KUKA KRL program: EPS_2_25694_BP02_A_20251117072356.src

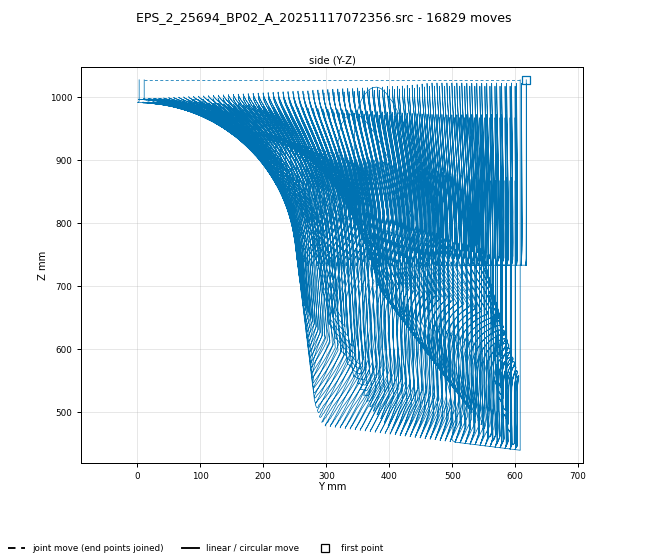
[picture p0: tool path of EPS_2_25694_BP02_A_20251117072356.src, 16829 of 16831 moves have a stored position in this frame; points joined in program order, loops and branches not executed]
&ACCESS RVP
&REL 4
&COMMENT QRS 19112012
&PARAM EDITMASK = *
DEF PART()
EXT BAS (BAS_COMMAND :IN,REAL :IN )
INT I
BAS (#INITMOV,0 )

;KUKA QRS Post kuka4.cps  Date:22-06-2017 !

File_ID=2911

QRS_PRE_INIT()

;Init var - Until changes are made in qrs_pre_init
Outlet_Square_prg=0
Inlet_1_Square_prg=0
Inlet_2_Square_prg=0
Inlet_3_Square_prg=0
Inlet_4_Square_prg=0
Inlet_5_Square_prg=0

Outlet_1={X 0.000, Y 466.000, Z 789.500, B 0.000, E1 0.000 }
Inlet_1={X 0.000, Y 466.000, Z 739.500, B 0.000, E1 180.000 }
Inlet_2={X 0.000, Y 537.940, Z 362.500, B 0.000, E1 273.000 }
Outlet_1_type=457
Inlet_1_type=457
Inlet_2_type=251
;QRS#1=Sidecore dimensions
;QRS#2=450-18" Concrete
;QRS#3=450-18" Concrete
;QRS#4=250-10" PVC SDR 35
;QRS#5=
;QRS#6=
;QRS#7=
;QRS#8=
;QRS#9=28A PSX-2
;QRS#10=28A PSX-2
;QRS#11=14M PSX
;QRS#12=
;QRS#13=
;QRS#14=
;QRS#15=
;QRS#16=1220x127x1372 4,5'
;QRS#17=EPS Height
;QRS#18=1018
;QRS#19=*
;QRS#20= UPDATED VERSION 22-06-2017
;QRS#21=*
Outlet_Square=0250
Inlet_1_Square=0250
Inlet_2_Square=0100
Inlet_3_Square=0
Inlet_4_Square=0
Inlet_5_Square=0
Mill_Square=1
Outlet_Square_Prg=274
Inlet_1_Square_prg=274
Inlet_2_Square_prg=205

QRS_INIT()

$ADVANCE=5

; T1
PTP {E1 171.215,E2 171.215}
PTP {X 0,Y 617.568,A -85,B 0,C 180,E1 171.215,E2 171.215,E3 0,E4 0,E5 0,E6 0}
QRS_SPEED_INIT()
LIN {X 0,Y 617.568,Z 1028,A -85,B 0,C 180,E1 171.215,E2 171.215,E3 0,E4 0,E5 0,E6 0} C_VEL
LIN {X 0,Y 617.568,Z 735.66,A -85,B 0,C 180,E1 171.215,E2 171.215} C_VEL
LIN {X 0,Y 617.546,Z 733.66,A -85,B 0,C 180,E1 171.401,E2 171.401} C_VEL
LIN {X 0,Y 617.995,Z 733.66,A -85,B 0,C 180,E1 174.214,E2 174.214} C_VEL
LIN {X 0,Y 618.056,Z 733.66,A -85,B 0,C 180,E1 178.845,E2 178.845} C_VEL
LIN {X 0,Y 618.024,Z 733.66,A -85,B 0,C 180,E1 183.468,E2 183.468} C_VEL
LIN {X 0,Y 618.034,Z 733.66,A -85,B 0,C 180,E1 188.114,E2 188.114} C_VEL
LIN {X 0,Y 618.015,Z 733.66,A -85,B 0,C 180,E1 192.815,E2 192.815} C_VEL
LIN {X 0,Y 617.991,Z 733.66,A -85,B 0,C 180,E1 197.606,E2 197.606} C_VEL
LIN {X 0,Y 617.8,Z 733.66,A -85,B 0,C 180,E1 198.557,E2 198.557} C_VEL
LIN {X 0,Y 617.948,Z 733.66,A -85,B 0,C 180,E1 202.529,E2 202.529} C_VEL
LIN {X 0,Y 617.447,Z 733.66,A -85,B 0,C 180,E1 205.076,E2 205.076} C_VEL
LIN {X 0,Y 617.888,Z 733.66,A -85,B 0,C 180,E1 207.636,E2 207.636} C_VEL
LIN {X 0,Y 617.379,Z 733.66,A -85,B 0,C 180,E1 210.305,E2 210.305} C_VEL
LIN {X 0,Y 617.845,Z 733.66,A -85,B 0,C 180,E1 212.995,E2 212.995} C_VEL
LIN {X 0,Y 617.716,Z 733.66,A -85,B 0,C 180,E1 214.198,E2 214.198} C_VEL
LIN {X 0,Y 617.779,Z 733.66,A -85,B 0,C 180,E1 218.705,E2 218.705} C_VEL
LIN {X 0,Y 617.447,Z 733.66,A -85,B 0,C 180,E1 221.76,E2 221.76} C_VEL
LIN {X 0,Y 617.88,Z 733.66,A -85,B 0,C 180,E1 224.901,E2 224.901} C_VEL
LIN {X 0,Y 617.778,Z 733.66,A -85,B 0,C 180,E1 228.274,E2 228.274} C_VEL
LIN {X 0,Y 617.563,Z 733.66,A -85,B 0,C 180,E1 231.279,E2 231.279} C_VEL
LIN {X 0,Y 617.589,Z 733.66,A -85,B 0,C 180,E1 231.899,E2 231.899} C_VEL
LIN {X 0,Y 617.834,Z 733.66,A -85,B 0,C 180,E1 234.203,E2 234.203} C_VEL
LIN {X 0,Y 617.355,Z 733.66,A -85,B 0,C 180,E1 236.976,E2 236.976} C_VEL
LIN {X 0,Y 617.906,Z 733.66,A -85,B 0,C 180,E1 239.724,E2 239.724} C_VEL
LIN {X 0,Y 617.897,Z 733.66,A -85,B 0,C 180,E1 243.987,E2 243.987} C_VEL
LIN {X 0,Y 617.787,Z 733.66,A -85,B 0,C 180,E1 244.426,E2 244.426} C_VEL
LIN {X 0,Y 617.131,Z 733.66,A -85,B 0,C 180,E1 244.544,E2 244.544} C_VEL
LIN {X 0,Y 616.404,Z 733.66,A -85,B 0,C 180,E1 244.615,E2 244.615} C_VEL
LIN {X 0,Y 617.534,Z 739.849,A -85,B 0,C 180,E1 244.745,E2 244.745} C_VEL
LIN {X 0,Y 617.679,Z 744.384,A -85,B 0,C 180,E1 244.809,E2 244.809} C_VEL
LIN {X 0,Y 617.925,Z 800.182,A -85,B 0,C 180,E1 245.528,E2 245.528} C_VEL
LIN {X 0,Y 617.874,Z 810.032,A -85,B 0,C 180,E1 245.684,E2 245.684} C_VEL
LIN {X 0,Y 617.799,Z 819.999,A -85,B 0,C 180,E1 245.88,E2 245.88} C_VEL
LIN {X 0,Y 617.89,Z 833.169,A -85,B 0,C 180,E1 246.218,E2 246.218} C_VEL
LIN {X 0,Y 617.827,Z 843.59,A -85,B 0,C 180,E1 246.528,E2 246.528} C_VEL
LIN {X 0,Y 617.931,Z 855.912,A -85,B 0,C 180,E1 246.969,E2 246.969} C_VEL
LIN {X 0,Y 617.951,Z 866.365,A -85,B 0,C 180,E1 247.393,E2 247.393} C_VEL
LIN {X 0,Y 617.873,Z 876.668,A -85,B 0,C 180,E1 247.859,E2 247.859} C_VEL
LIN {X 0,Y 617.944,Z 887.338,A -85,B 0,C 180,E1 248.406,E2 248.406} C_VEL
LIN {X 0,Y 617.966,Z 898.213,A -85,B 0,C 180,E1 249.027,E2 249.027} C_VEL
LIN {X 0,Y 617.938,Z 908.022,A -85,B 0,C 180,E1 249.643,E2 249.643} C_VEL
LIN {X 0,Y 617.949,Z 917.528,A -85,B 0,C 180,E1 250.301,E2 250.301} C_VEL
LIN {X 0,Y 617.957,Z 926.721,A -85,B 0,C 180,E1 250.999,E2 250.999} C_VEL
LIN {X 0,Y 617.963,Z 935.648,A -85,B 0,C 180,E1 251.739,E2 251.739} C_VEL
LIN {X 0,Y 617.942,Z 944.029,A -85,B 0,C 180,E1 252.497,E2 252.497} C_VEL
LIN {X 0,Y 617.896,Z 951.424,A -85,B 0,C 180,E1 253.221,E2 253.221} C_VEL
LIN {X 0,Y 617.949,Z 959.127,A -85,B 0,C 180,E1 254.046,E2 254.046} C_VEL
LIN {X 0,Y 617.972,Z 965.662,A -85,B 0,C 180,E1 254.803,E2 254.803} C_VEL
LIN {X 0,Y 617.889,Z 972.774,A -85,B 0,C 180,E1 255.697,E2 255.697} C_VEL
LIN {X 0,Y 617.879,Z 979.238,A -85,B 0,C 180,E1 256.589,E2 256.589} C_VEL
LIN {X 0,Y 617.985,Z 985.097,A -85,B 0,C 180,E1 257.481,E2 257.481} C_VEL
LIN {X 0,Y 617.89,Z 990.459,A -85,B 0,C 180,E1 258.365,E2 258.365} C_VEL
LIN {X 0,Y 617.834,Z 996.765,A -85,B 0,C 180,E1 259.542,E2 259.542} C_VEL
LIN {X 0,Y 617.91,Z 1000.345,A -85,B 0,C 180,E1 260.284,E2 260.284} C_VEL
LIN {X 0,Y 617.922,Z 1005.379,A -85,B 0,C 180,E1 261.454,E2 261.454} C_VEL
LIN {X 0,Y 617.827,Z 1008.757,A -85,B 0,C 180,E1 262.35,E2 262.35} C_VEL
LIN {X 0,Y 617.939,Z 1013.149,A -85,B 0,C 180,E1 263.748,E2 263.748} C_VEL
LIN {X 0,Y 617.916,Z 1015.616,A -85,B 0,C 180,E1 264.677,E2 264.677} C_VEL
LIN {X 0,Y 617.776,Z 1018.488,A -85,B 0,C 180,E1 266.068,E2 266.068} C_VEL
LIN {X 0,Y 617.811,Z 1019.258,A -85,B 0,C 180,E1 266.531,E2 266.531} C_VEL
LIN {X 0,Y 617.947,Z 1020.966,A -85,B 0,C 180,E1 267.92,E2 267.92} C_VEL
LIN {X 0,Y 617.797,Z 1021.661,A -85,B 0,C 180,E1 268.844,E2 268.844} C_VEL
LIN {X 0,Y 617.834,Z 1021.908,A -85,B 0,C 180,E1 270.231,E2 270.231} C_VEL
LIN {X 0,Y 617.983,Z 1021.61,A -85,B 0,C 180,E1 271.156,E2 271.156} C_VEL
LIN {X 0,Y 617.821,Z 1020.474,A -85,B 0,C 180,E1 272.543,E2 272.543} C_VEL
LIN {X 0,Y 617.856,Z 1019.246,A -85,B 0,C 180,E1 273.469,E2 273.469} C_VEL
LIN {X 0,Y 618.001,Z 1017.612,A -85,B 0,C 180,E1 274.395,E2 274.395} C_VEL
LIN {X 0,Y 617.856,Z 1015.632,A -85,B 0,C 180,E1 275.323,E2 275.323} C_VEL
LIN {X 0,Y 617.792,Z 1013.186,A -85,B 0,C 180,E1 276.253,E2 276.253} C_VEL
LIN {X 0,Y 617.955,Z 1008.725,A -85,B 0,C 180,E1 277.648,E2 277.648} C_VEL
LIN {X 0,Y 617.882,Z 1004.324,A -85,B 0,C 180,E1 278.801,E2 278.801} C_VEL
LIN {X 0,Y 617.827,Z 1000.605,A -85,B 0,C 180,E1 279.668,E2 279.668} C_VEL
LIN {X 0,Y 617.937,Z 995.255,A -85,B 0,C 180,E1 280.751,E2 280.751} C_VEL
LIN {X 0,Y 617.942,Z 990.447,A -85,B 0,C 180,E1 281.634,E2 281.634} C_VEL
LIN {X 0,Y 617.864,Z 983.196,A -85,B 0,C 180,E1 282.818,E2 282.818} C_VEL
LIN {X 0,Y 617.94,Z 977.134,A -85,B 0,C 180,E1 283.707,E2 283.707} C_VEL
LIN {X 0,Y 617.957,Z 970.467,A -85,B 0,C 180,E1 284.6,E2 284.6} C_VEL
LIN {X 0,Y 617.883,Z 962.504,A -85,B 0,C 180,E1 285.571,E2 285.571} C_VEL
LIN {X 0,Y 617.918,Z 955.447,A -85,B 0,C 180,E1 286.357,E2 286.357} C_VEL
LIN {X 0,Y 617.97,Z 947.287,A -85,B 0,C 180,E1 287.188,E2 287.188} C_VEL
LIN {X 0,Y 617.932,Z 940.146,A -85,B 0,C 180,E1 287.864,E2 287.864} C_VEL
LIN {X 0,Y 617.923,Z 931.257,A -85,B 0,C 180,E1 288.634,E2 288.634} C_VEL
LIN {X 0,Y 617.943,Z 922.354,A -85,B 0,C 180,E1 289.339,E2 289.339} C_VEL
LIN {X 0,Y 617.96,Z 913.855,A -85,B 0,C 180,E1 289.959,E2 289.959} C_VEL
LIN {X 0,Y 617.948,Z 904.462,A -85,B 0,C 180,E1 290.588,E2 290.588} C_VEL
LIN {X 0,Y 617.918,Z 894.269,A -85,B 0,C 180,E1 291.207,E2 291.207} C_VEL
LIN {X 0,Y 617.943,Z 884.404,A -85,B 0,C 180,E1 291.749,E2 291.749} C_VEL
LIN {X 0,Y 617.959,Z 873.347,A -85,B 0,C 180,E1 292.294,E2 292.294} C_VEL
LIN {X 0,Y 617.927,Z 862.59,A -85,B 0,C 180,E1 292.768,E2 292.768} C_VEL
LIN {X 0,Y 617.804,Z 852.699,A -85,B 0,C 180,E1 293.16,E2 293.16} C_VEL
LIN {X 0,Y 617.934,Z 839.476,A -85,B 0,C 180,E1 293.596,E2 293.596} C_VEL
LIN {X 0,Y 617.909,Z 828.006,A -85,B 0,C 180,E1 293.92,E2 293.92} C_VEL
LIN {X 0,Y 617.764,Z 816.647,A -85,B 0,C 180,E1 294.191,E2 294.191} C_VEL
LIN {X 0,Y 617.917,Z 805.001,A -85,B 0,C 180,E1 294.401,E2 294.401} C_VEL
LIN {X 0,Y 617.885,Z 787.363,A -85,B 0,C 180,E1 294.643,E2 294.643} C_VEL
LIN {X 0,Y 617.595,Z 740.263,A -85,B 0,C 180,E1 295.247,E2 295.247} C_VEL
LIN {X 0,Y 616.482,Z 734.086,A -85,B 0,C 180,E1 295.374,E2 295.374} C_VEL
LIN {X 0,Y 616.463,Z 733.66,A -85,B 0,C 180,E1 295.391,E2 295.391} C_VEL
LIN {X 0,Y 616.669,Z 733.66,A -85,B 0,C 180,E1 295.406,E2 295.406} C_VEL
LIN {X 0,Y 618.016,Z 733.66,A -85,B 0,C 180,E1 295.712,E2 295.712} C_VEL
LIN {X 0,Y 617.906,Z 733.66,A -85,B 0,C 180,E1 300.277,E2 300.277} C_VEL
LIN {X 0,Y 617.354,Z 733.66,A -85,B 0,C 180,E1 303.025,E2 303.025} C_VEL
LIN {X 0,Y 617.832,Z 733.66,A -85,B 0,C 180,E1 305.797,E2 305.797} C_VEL
LIN {X 0,Y 617.565,Z 733.66,A -85,B 0,C 180,E1 308.721,E2 308.721} C_VEL
LIN {X 0,Y 617.776,Z 733.66,A -85,B 0,C 180,E1 311.732,E2 311.732} C_VEL
LIN {X 0,Y 617.882,Z 733.66,A -85,B 0,C 180,E1 315.1,E2 315.1} C_VEL
LIN {X 0,Y 617.453,Z 733.66,A -85,B 0,C 180,E1 318.308,E2 318.308} C_VEL
LIN {X 0,Y 617.785,Z 733.66,A -85,B 0,C 180,E1 321.296,E2 321.296} C_VEL
LIN {X 0,Y 617.728,Z 733.66,A -85,B 0,C 180,E1 325.801,E2 325.801} C_VEL
LIN {X 0,Y 617.883,Z 733.66,A -85,B 0,C 180,E1 327.007,E2 327.007} C_VEL
LIN {X 0,Y 617.633,Z 733.66,A -85,B 0,C 180,E1 330.177,E2 330.177} C_VEL
LIN {X 0,Y 617.638,Z 733.66,A -85,B 0,C 180,E1 332.352,E2 332.352} C_VEL
LIN {X 0,Y 617.494,Z 733.66,A -85,B 0,C 180,E1 335.247,E2 335.247} C_VEL
LIN {X 0,Y 617.713,Z 733.66,A -85,B 0,C 180,E1 337.462,E2 337.462} C_VEL
LIN {X 0,Y 617.768,Z 733.66,A -85,B 0,C 180,E1 341.453,E2 341.453} C_VEL
LIN {X 0,Y 617.438,Z 733.66,A -85,B 0,C 180,E1 342.378,E2 342.378} C_VEL
LIN {X 0,Y 617.027,Z 733.66,A -85,B 0,C 180,E1 342.43,E2 342.43} C_VEL
LIN {X 0,Y 617.816,Z 744.735,A -85,B 0,C 180,E1 342.612,E2 342.612} C_VEL
LIN {X 0,Y 617.988,Z 754.107,A -85,B 0,C 180,E1 342.807,E2 342.807} C_VEL
LIN {X 0,Y 618.017,Z 763.539,A -85,B 0,C 180,E1 343.055,E2 343.055} C_VEL
LIN {X 0,Y 617.945,Z 772.657,A -85,B 0,C 180,E1 343.357,E2 343.357} C_VEL
LIN {X 0,Y 618.019,Z 781.507,A -85,B 0,C 180,E1 343.712,E2 343.712} C_VEL
LIN {X 0,Y 618.022,Z 791.359,A -85,B 0,C 180,E1 344.179,E2 344.179} C_VEL
LIN {X 0,Y 617.995,Z 798.507,A -85,B 0,C 180,E1 344.573,E2 344.573} C_VEL
LIN {X 0,Y 618.012,Z 805.794,A -85,B 0,C 180,E1 345.028,E2 345.028} C_VEL
LIN {X 0,Y 618.02,Z 813.252,A -85,B 0,C 180,E1 345.551,E2 345.551} C_VEL
LIN {X 0,Y 618.001,Z 820.673,A -85,B 0,C 180,E1 346.146,E2 346.146} C_VEL
LIN {X 0,Y 617.998,Z 827.267,A -85,B 0,C 180,E1 346.74,E2 346.74} C_VEL
LIN {X 0,Y 617.988,Z 834.495,A -85,B 0,C 180,E1 347.481,E2 347.481} C_VEL
LIN {X 0,Y 617.999,Z 840.799,A -85,B 0,C 180,E1 348.22,E2 348.22} C_VEL
LIN {X 0,Y 617.966,Z 846.334,A -85,B 0,C 180,E1 348.956,E2 348.956} C_VEL
LIN {X 0,Y 617.958,Z 851.386,A -85,B 0,C 180,E1 349.732,E2 349.732} C_VEL
LIN {X 0,Y 617.992,Z 855.679,A -85,B 0,C 180,E1 350.486,E2 350.486} C_VEL
LIN {X 0,Y 617.971,Z 858.976,A -85,B 0,C 180,E1 351.146,E2 351.146} C_VEL
LIN {X 0,Y 617.919,Z 862.179,A -85,B 0,C 180,E1 351.885,E2 351.885} C_VEL
LIN {X 0,Y 617.964,Z 865.461,A -85,B 0,C 180,E1 352.818,E2 352.818} C_VEL
LIN {X 0,Y 617.965,Z 868.095,A -85,B 0,C 180,E1 353.749,E2 353.749} C_VEL
LIN {X 0,Y 617.919,Z 869.981,A -85,B 0,C 180,E1 354.677,E2 354.677} C_VEL
LIN {X 0,Y 617.982,Z 871.236,A -85,B 0,C 180,E1 355.605,E2 355.605} C_VEL
LIN {X 0,Y 617.939,Z 871.836,A -85,B 0,C 180,E1 356.532,E2 356.532} C_VEL
LIN {X 0,Y 617.919,Z 871.824,A -85,B 0,C 180,E1 357.457,E2 357.457} C_VEL
LIN {X 0,Y 617.957,Z 871.548,A -85,B 0,C 180,E1 357.92,E2 357.92} C_VEL
LIN {X 0,Y 617.981,Z 870.597,A -85,B 0,C 180,E1 358.845,E2 358.845} C_VEL
LIN {X 0,Y 617.919,Z 868.964,A -85,B 0,C 180,E1 359.769,E2 359.769} C_VEL
LIN {X 0,Y 617.931,Z 867.927,A -85,B 0,C 180,E1 360.231,E2 360.231} C_VEL
LIN {X 0,Y 617.995,Z 865.25,A -85,B 0,C 180,E1 361.155,E2 361.155} C_VEL
LIN {X 0,Y 617.929,Z 861.961,A -85,B 0,C 180,E1 362.08,E2 362.08} C_VEL
LIN {X 0,Y 617.948,Z 857.807,A -85,B 0,C 180,E1 363.005,E2 363.005} C_VEL
LIN {X 0,Y 618.008,Z 852.875,A -85,B 0,C 180,E1 363.931,E2 363.931} C_VEL
LIN {X 0,Y 617.968,Z 848.545,A -85,B 0,C 180,E1 364.627,E2 364.627} C_VEL
LIN {X 0,Y 617.969,Z 843.641,A -85,B 0,C 180,E1 365.322,E2 365.322} C_VEL
LIN {X 0,Y 617.995,Z 838.117,A -85,B 0,C 180,E1 366.019,E2 366.019} C_VEL
LIN {X 0,Y 617.998,Z 831.807,A -85,B 0,C 180,E1 366.716,E2 366.716} C_VEL
LIN {X 0,Y 617.991,Z 825.901,A -85,B 0,C 180,E1 367.298,E2 367.298} C_VEL
LIN {X 0,Y 618.018,Z 819.311,A -85,B 0,C 180,E1 367.881,E2 367.881} C_VEL
LIN {X 0,Y 618.024,Z 811.759,A -85,B 0,C 180,E1 368.467,E2 368.467} C_VEL
LIN {X 0,Y 618.012,Z 804.455,A -85,B 0,C 180,E1 368.97,E2 368.97} C_VEL
LIN {X 0,Y 618.008,Z 796.87,A -85,B 0,C 180,E1 369.433,E2 369.433} C_VEL
LIN {X 0,Y 618.017,Z 788.03,A -85,B 0,C 180,E1 369.898,E2 369.898} C_VEL
LIN {X 0,Y 618.03,Z 779.833,A -85,B 0,C 180,E1 370.269,E2 370.269} C_VEL
LIN {X 0,Y 618.017,Z 770.184,A -85,B 0,C 180,E1 370.641,E2 370.641} C_VEL
LIN {X 0,Y 617.996,Z 761.871,A -85,B 0,C 180,E1 370.902,E2 370.902} C_VEL
LIN {X 0,Y 618.051,Z 752.155,A -85,B 0,C 180,E1 371.146,E2 371.146} C_VEL
LIN {X 0,Y 618.03,Z 743.677,A -85,B 0,C 180,E1 371.312,E2 371.312} C_VEL
LIN {X 0,Y 617.969,Z 738.905,A -85,B 0,C 180,E1 371.382,E2 371.382} C_VEL
LIN {X 0,Y 617.381,Z 735.038,A -85,B 0,C 180,E1 371.448,E2 371.448} C_VEL
LIN {X 0,Y 617.223,Z 733.66,A -85,B 0,C 180,E1 371.506,E2 371.506} C_VEL
LIN {X 0,Y 618.074,Z 733.66,A -85,B 0,C 180,E1 371.931,E2 371.931} C_VEL
LIN {X 0,Y 617.858,Z 733.66,A -85,B 0,C 180,E1 372.818,E2 372.818} C_VEL
LIN {X 0,Y 617.953,Z 733.66,A -85,B 0,C 180,E1 377.607,E2 377.607} C_VEL
LIN {X 0,Y 617.769,Z 733.66,A -85,B 0,C 180,E1 378.547,E2 378.547} C_VEL
LIN {X 0,Y 617.917,Z 733.66,A -85,B 0,C 180,E1 382.53,E2 382.53} C_VEL
LIN {X 0,Y 617.429,Z 733.66,A -85,B 0,C 180,E1 385.077,E2 385.077} C_VEL
LIN {X 0,Y 617.885,Z 733.66,A -85,B 0,C 180,E1 387.636,E2 387.636} C_VEL
LIN {X 0,Y 617.381,Z 733.66,A -85,B 0,C 180,E1 390.305,E2 390.305} C_VEL
LIN {X 0,Y 617.86,Z 733.66,A -85,B 0,C 180,E1 392.994,E2 392.994} C_VEL
LIN {X 0,Y 617.717,Z 733.66,A -85,B 0,C 180,E1 394.198,E2 394.198} C_VEL
LIN {X 0,Y 617.788,Z 733.66,A -85,B 0,C 180,E1 398.704,E2 398.704} C_VEL
LIN {X 0,Y 617.449,Z 733.66,A -85,B 0,C 180,E1 401.76,E2 401.76} C_VEL
LIN {X 0,Y 617.885,Z 733.66,A -85,B 0,C 180,E1 404.9,E2 404.9} C_VEL
LIN {X 0,Y 617.79,Z 733.66,A -85,B 0,C 180,E1 408.273,E2 408.273} C_VEL
LIN {X 0,Y 617.55,Z 733.66,A -85,B 0,C 180,E1 411.278,E2 411.278} C_VEL
LIN {X 0,Y 617.572,Z 733.66,A -85,B 0,C 180,E1 411.901,E2 411.901} C_VEL
LIN {X 0,Y 617.803,Z 733.66,A -85,B 0,C 180,E1 414.201,E2 414.201} C_VEL
LIN {X 0,Y 617.341,Z 733.66,A -85,B 0,C 180,E1 416.975,E2 416.975} C_VEL
LIN {X 0,Y 617.87,Z 733.66,A -85,B 0,C 180,E1 419.721,E2 419.721} C_VEL
LIN {X 0,Y 618.08,Z 733.66,A -85,B 0,C 180,E1 424.951,E2 424.951} C_VEL
LIN {X 0,Y 617.2,Z 733.66,A -85,B 0,C 180,E1 425.214,E2 425.214} C_VEL
LIN {X 0,Y 617.09,Z 733.66,A -85,B 0,C 180,E1 425.227,E2 425.227} C_VEL
LIN {X 0,Y 617.703,Z 736.777,A -85,B 0,C 180,E1 425.297,E2 425.297} C_VEL
LIN {X 0,Y 617.723,Z 754.51,A -85,B 0,C 180,E1 425.539,E2 425.539} C_VEL
LIN {X 0,Y 617.86,Z 764.098,A -85,B 0,C 180,E1 425.718,E2 425.718} C_VEL
LIN {X 0,Y 617.907,Z 773.477,A -85,B 0,C 180,E1 425.924,E2 425.924} C_VEL
LIN {X 0,Y 617.865,Z 783.691,A -85,B 0,C 180,E1 426.187,E2 426.187} C_VEL
LIN {X 0,Y 617.854,Z 792.887,A -85,B 0,C 180,E1 426.46,E2 426.46} C_VEL
LIN {X 0,Y 617.949,Z 804.75,A -85,B 0,C 180,E1 426.879,E2 426.879} C_VEL
LIN {X 0,Y 617.922,Z 815.627,A -85,B 0,C 180,E1 427.313,E2 427.313} C_VEL
LIN {X 0,Y 617.904,Z 826.006,A -85,B 0,C 180,E1 427.782,E2 427.782} C_VEL
LIN {X 0,Y 617.948,Z 838.136,A -85,B 0,C 180,E1 428.406,E2 428.406} C_VEL
LIN {X 0,Y 617.938,Z 848.936,A -85,B 0,C 180,E1 429.026,E2 429.026} C_VEL
LIN {X 0,Y 617.922,Z 858.679,A -85,B 0,C 180,E1 429.643,E2 429.643} C_VEL
LIN {X 0,Y 617.947,Z 868.08,A -85,B 0,C 180,E1 430.297,E2 430.297} C_VEL
LIN {X 0,Y 617.965,Z 877.14,A -85,B 0,C 180,E1 430.988,E2 430.988} C_VEL
LIN {X 0,Y 617.959,Z 886.054,A -85,B 0,C 180,E1 431.73,E2 431.73} C_VEL
LIN {X 0,Y 617.941,Z 893.416,A -85,B 0,C 180,E1 432.393,E2 432.393} C_VEL
LIN {X 0,Y 617.929,Z 901.731,A -85,B 0,C 180,E1 433.21,E2 433.21} C_VEL
LIN {X 0,Y 617.984,Z 909.303,A -85,B 0,C 180,E1 434.023,E2 434.023} C_VEL
LIN {X 0,Y 617.922,Z 916.028,A -85,B 0,C 180,E1 434.801,E2 434.801} C_VEL
LIN {X 0,Y 617.883,Z 923.102,A -85,B 0,C 180,E1 435.697,E2 435.697} C_VEL
LIN {X 0,Y 617.954,Z 929.522,A -85,B 0,C 180,E1 436.591,E2 436.591} C_VEL
LIN {X 0,Y 617.932,Z 935.377,A -85,B 0,C 180,E1 437.48,E2 437.48} C_VEL
LIN {X 0,Y 617.834,Z 940.721,A -85,B 0,C 180,E1 438.364,E2 438.364} C_VEL
LIN {X 0,Y 617.882,Z 946.971,A -85,B 0,C 180,E1 439.542,E2 439.542} C_VEL
LIN {X 0,Y 617.995,Z 950.749,A -85,B 0,C 180,E1 440.329,E2 440.329} C_VEL
LIN {X 0,Y 617.842,Z 955.587,A -85,B 0,C 180,E1 441.458,E2 441.458} C_VEL
LIN {X 0,Y 617.843,Z 958.922,A -85,B 0,C 180,E1 442.35,E2 442.35} C_VEL
LIN {X 0,Y 617.961,Z 961.91,A -85,B 0,C 180,E1 443.283,E2 443.283} C_VEL
LIN {X 0,Y 617.885,Z 964.529,A -85,B 0,C 180,E1 444.212,E2 444.212} C_VEL
LIN {X 0,Y 617.792,Z 966.751,A -85,B 0,C 180,E1 445.14,E2 445.14} C_VEL
LIN {X 0,Y 617.804,Z 967.762,A -85,B 0,C 180,E1 445.604,E2 445.604} C_VEL
LIN {X 0,Y 617.919,Z 969.305,A -85,B 0,C 180,E1 446.531,E2 446.531} C_VEL
LIN {X 0,Y 617.942,Z 970.495,A -85,B 0,C 180,E1 447.457,E2 447.457} C_VEL
LIN {X 0,Y 617.799,Z 971.692,A -85,B 0,C 180,E1 448.844,E2 448.844} C_VEL
LIN {X 0,Y 617.859,Z 971.913,A -85,B 0,C 180,E1 449.769,E2 449.769} C_VEL
LIN {X 0,Y 617.971,Z 971.75,A -85,B 0,C 180,E1 450.693,E2 450.693} C_VEL
LIN {X 0,Y 617.912,Z 971.597,A -85,B 0,C 180,E1 451.155,E2 451.155} C_VEL
LIN {X 0,Y 617.83,Z 970.962,A -85,B 0,C 180,E1 452.08,E2 452.08} C_VEL
LIN {X 0,Y 617.944,Z 969.146,A -85,B 0,C 180,E1 453.468,E2 453.468} C_VEL
LIN {X 0,Y 617.98,Z 968.359,A -85,B 0,C 180,E1 453.931,E2 453.931} C_VEL
LIN {X 0,Y 617.794,Z 965.548,A -85,B 0,C 180,E1 455.324,E2 455.324} C_VEL
LIN {X 0,Y 617.823,Z 963.059,A -85,B 0,C 180,E1 456.253,E2 456.253} C_VEL
LIN {X 0,Y 617.953,Z 960.131,A -85,B 0,C 180,E1 457.182,E2 457.182} C_VEL
LIN {X 0,Y 617.871,Z 956.83,A -85,B 0,C 180,E1 458.116,E2 458.116} C_VEL
LIN {X 0,Y 617.817,Z 953.947,A -85,B 0,C 180,E1 458.848,E2 458.848} C_VEL
LIN {X 0,Y 617.861,Z 950.456,A -85,B 0,C 180,E1 459.652,E2 459.652} C_VEL
LIN {X 0,Y 617.954,Z 945.008,A -85,B 0,C 180,E1 460.75,E2 460.75} C_VEL
LIN {X 0,Y 617.849,Z 940.205,A -85,B 0,C 180,E1 461.636,E2 461.636} C_VEL
LIN {X 0,Y 617.826,Z 934.857,A -85,B 0,C 180,E1 462.522,E2 462.522} C_VEL
LIN {X 0,Y 617.972,Z 926.799,A -85,B 0,C 180,E1 463.706,E2 463.706} C_VEL
LIN {X 0,Y 617.922,Z 920.112,A -85,B 0,C 180,E1 464.601,E2 464.601} C_VEL
LIN {X 0,Y 617.89,Z 913.695,A -85,B 0,C 180,E1 465.39,E2 465.39} C_VEL
LIN {X 0,Y 617.959,Z 904.86,A -85,B 0,C 180,E1 466.371,E2 466.371} C_VEL
LIN {X 0,Y 617.967,Z 897.837,A -85,B 0,C 180,E1 467.09,E2 467.09} C_VEL
LIN {X 0,Y 617.938,Z 889.57,A -85,B 0,C 180,E1 467.869,E2 467.869} C_VEL
LIN {X 0,Y 617.955,Z 881.128,A -85,B 0,C 180,E1 468.598,E2 468.598} C_VEL
LIN {X 0,Y 617.959,Z 872.754,A -85,B 0,C 180,E1 469.264,E2 469.264} C_VEL
LIN {X 0,Y 617.953,Z 863.173,A -85,B 0,C 180,E1 469.961,E2 469.961} C_VEL
LIN {X 0,Y 617.937,Z 853.736,A -85,B 0,C 180,E1 470.588,E2 470.588} C_VEL
LIN {X 0,Y 617.88,Z 843.468,A -85,B 0,C 180,E1 471.208,E2 471.208} C_VEL
LIN {X 0,Y 617.941,Z 833.513,A -85,B 0,C 180,E1 471.749,E2 471.749} C_VEL
LIN {X 0,Y 617.936,Z 824.09,A -85,B 0,C 180,E1 472.217,E2 472.217} C_VEL
LIN {X 0,Y 617.817,Z 812.471,A -85,B 0,C 180,E1 472.732,E2 472.732} C_VEL
LIN {X 0,Y 617.956,Z 800.776,A -85,B 0,C 180,E1 473.175,E2 473.175} C_VEL
LIN {X 0,Y 617.937,Z 789.271,A -85,B 0,C 180,E1 473.557,E2 473.557} C_VEL
LIN {X 0,Y 617.803,Z 778.065,A -85,B 0,C 180,E1 473.878,E2 473.878} C_VEL
LIN {X 0,Y 617.931,Z 766.646,A -85,B 0,C 180,E1 474.139,E2 474.139} C_VEL
LIN {X 0,Y 617.94,Z 754.847,A -85,B 0,C 180,E1 474.357,E2 474.357} C_VEL
LIN {X 0,Y 617.715,Z 736.943,A -85,B 0,C 180,E1 474.61,E2 474.61} C_VEL
LIN {X 0,Y 617.665,Z 733.66,A -85,B 0,C 180,E1 474.655,E2 474.655} C_VEL
LIN {X 0,Y 618.06,Z 733.66,A -85,B 0,C 180,E1 474.797,E2 474.797} C_VEL
LIN {X 0,Y 617.954,Z 733.66,A -85,B 0,C 180,E1 477.633,E2 477.633} C_VEL
LIN {X 0,Y 617.376,Z 733.66,A -85,B 0,C 180,E1 480.305,E2 480.305} C_VEL
LIN {X 0,Y 617.848,Z 733.66,A -85,B 0,C 180,E1 482.995,E2 482.995} C_VEL
LIN {X 0,Y 617.718,Z 733.66,A -85,B 0,C 180,E1 484.198,E2 484.198} C_VEL
LIN {X 0,Y 617.788,Z 733.66,A -85,B 0,C 180,E1 488.704,E2 488.704} C_VEL
LIN {X 0,Y 617.434,Z 733.66,A -85,B 0,C 180,E1 491.76,E2 491.76} C_VEL
LIN {X 0,Y 617.836,Z 733.66,A -85,B 0,C 180,E1 494.904,E2 494.904} C_VEL
LIN {X 0,Y 617.761,Z 733.66,A -85,B 0,C 180,E1 498.275,E2 498.275} C_VEL
LIN {X 0,Y 617.558,Z 733.66,A -85,B 0,C 180,E1 501.279,E2 501.279} C_VEL
LIN {X 0,Y 617.836,Z 733.66,A -85,B 0,C 180,E1 504.203,E2 504.203} C_VEL
LIN {X 0,Y 617.329,Z 733.66,A -85,B 0,C 180,E1 506.974,E2 506.974} C_VEL
LIN {X 0,Y 617.85,Z 733.66,A -85,B 0,C 180,E1 509.72,E2 509.72} C_VEL
LIN {X 0,Y 617.412,Z 733.66,A -85,B 0,C 180,E1 512.341,E2 512.341} C_VEL
LIN {X 0,Y 617.928,Z 733.66,A -85,B 0,C 180,E1 514.945,E2 514.945} C_VEL
LIN {X 0,Y 617.476,Z 733.66,A -85,B 0,C 180,E1 517.453,E2 517.453} C_VEL
LIN {X 0,Y 617.979,Z 733.66,A -85,B 0,C 180,E1 519.952,E2 519.952} C_VEL
LIN {X 0,Y 618.039,Z 733.66,A -85,B 0,C 180,E1 523.63,E2 523.63} C_VEL
LIN {X 0,Y 618.007,Z 733.66,A -85,B 0,C 180,E1 529.544,E2 529.544} C_VEL
LIN {X 0,Y 617.546,Z 733.66,A -85,B 0,C 180,E1 531.401,E2 531.401} C_VEL
LIN {X 0,Y 613.849,Z 733.66,A -85,B 0,C 180,E1 532.992,E2 532.992} C_VEL
LIN {X 0,Y 609.948,Z 733.66,A -85,B 0,C 180,E1 534.603,E2 534.603} C_VEL
LIN {X 0,Y 609.797,Z 733.66,A -85,B 0,C 180,E1 539.997,E2 539.997} C_VEL
LIN {X 0,Y 609.862,Z 733.66,A -85,B 0,C 180,E1 544.268,E2 544.268} C_VEL
LIN {X 0,Y 609.959,Z 733.66,A -85,B 0,C 180,E1 548.562,E2 548.562} C_VEL
LIN {X 0,Y 610.085,Z 733.66,A -85,B 0,C 180,E1 552.902,E2 552.902} C_VEL
LIN {X 0,Y 609.84,Z 733.66,A -85,B 0,C 180,E1 558.825,E2 558.825} C_VEL
LIN {X 0,Y 609.743,Z 733.66,A -85,B 0,C 180,E1 563.405,E2 563.405} C_VEL
LIN {X 0,Y 609.805,Z 733.66,A -85,B 0,C 180,E1 568.143,E2 568.143} C_VEL
LIN {X 0,Y 609.95,Z 733.66,A -85,B 0,C 180,E1 573.095,E2 573.095} C_VEL
LIN {X 0,Y 609.605,Z 733.66,A -85,B 0,C 180,E1 579.65,E2 579.65} C_VEL
LIN {X 0,Y 609.728,Z 733.66,A -85,B 0,C 180,E1 585.948,E2 585.948} C_VEL
LIN {X 0,Y 609.563,Z 733.66,A -85,B 0,C 180,E1 590.346,E2 590.346} C_VEL
LIN {X 0,Y 609.619,Z 733.66,A -85,B 0,C 180,E1 595.163,E2 595.163} C_VEL
LIN {X 0,Y 609.807,Z 733.66,A -85,B 0,C 180,E1 600.332,E2 600.332} C_VEL
LIN {X 0,Y 609.393,Z 733.66,A -85,B 0,C 180,E1 604.276,E2 604.276} C_VEL
LIN {X 0,Y 610.599,Z 758.456,A -85,B 0,C 180,E1 604.675,E2 604.675} C_VEL
LIN {X 0,Y 610.572,Z 821.161,A -85,B 0,C 180,E1 605.604,E2 605.604} C_VEL
LIN {X 0,Y 610.588,Z 857.058,A -85,B 0,C 180,E1 606.721,E2 606.721} C_VEL
LIN {X 0,Y 610.478,Z 891.255,A -85,B 0,C 180,E1 608.35,E2 608.35} C_VEL
LIN {X 0,Y 610.357,Z 924.126,A -85,B 0,C 180,E1 610.543,E2 610.543} C_VEL
LIN {X 0,Y 610.178,Z 951.986,A -85,B 0,C 180,E1 613.048,E2 613.048} C_VEL
LIN {X 0,Y 610.1,Z 976.637,A -85,B 0,C 180,E1 615.997,E2 615.997} C_VEL
LIN {X 0,Y 610.05,Z 994.768,A -85,B 0,C 180,E1 618.91,E2 618.91} C_VEL
LIN {X 0,Y 610.026,Z 1009.174,A -85,B 0,C 180,E1 622.154,E2 622.154} C_VEL
LIN {X 0,Y 610.028,Z 1017.451,A -85,B 0,C 180,E1 625.016,E2 625.016} C_VEL
LIN {X 0,Y 610.02,Z 1022.507,A -85,B 0,C 180,E1 628.578,E2 628.578} C_VEL
LIN {X 0,Y 610.116,Z 1022.507,A -85,B 0,C 180,E1 631.422,E2 631.422} C_VEL
LIN {X 0,Y 610.068,Z 1017.452,A -85,B 0,C 180,E1 634.983,E2 634.983} C_VEL
LIN {X 0,Y 610.086,Z 1006.497,A -85,B 0,C 180,E1 638.563,E2 638.563} C_VEL
LIN {X 0,Y 610.103,Z 989.709,A -85,B 0,C 180,E1 641.996,E2 641.996} C_VEL
LIN {X 0,Y 610.173,Z 968.258,A -85,B 0,C 180,E1 645.103,E2 645.103} C_VEL
LIN {X 0,Y 610.253,Z 941.577,A -85,B 0,C 180,E1 647.974,E2 647.974} C_VEL
LIN {X 0,Y 610.395,Z 910.989,A -85,B 0,C 180,E1 650.415,E2 650.415} C_VEL
LIN {X 0,Y 610.534,Z 878.716,A -85,B 0,C 180,E1 652.317,E2 652.317} C_VEL
LIN {X 0,Y 610.65,Z 843.322,A -85,B 0,C 180,E1 653.774,E2 653.774} C_VEL
LIN {X 0,Y 610.719,Z 806.699,A -85,B 0,C 180,E1 654.682,E2 654.682} C_VEL
LIN {X 0,Y 609.809,Z 737.78,A -85,B 0,C 180,E1 655.624,E2 655.624} C_VEL
LIN {X 0,Y 609.661,Z 733.66,A -85,B 0,C 180,E1 655.76,E2 655.76} C_VEL
LIN {X 0,Y 609.836,Z 733.66,A -85,B 0,C 180,E1 659.772,E2 659.772} C_VEL
LIN {X 0,Y 609.732,Z 733.66,A -85,B 0,C 180,E1 666.582,E2 666.582} C_VEL
LIN {X 0,Y 609.784,Z 733.66,A -85,B 0,C 180,E1 672.098,E2 672.098} C_VEL
LIN {X 0,Y 609.512,Z 733.66,A -85,B 0,C 180,E1 677.885,E2 677.885} C_VEL
LIN {X 0,Y 609.482,Z 733.66,A -85,B 0,C 180,E1 682.651,E2 682.651} C_VEL
LIN {X 0,Y 609.824,Z 733.66,A -85,B 0,C 180,E1 687.582,E2 687.582} C_VEL
LIN {X 0,Y 609.676,Z 733.66,A -85,B 0,C 180,E1 691.851,E2 691.851} C_VEL
LIN {X 0,Y 609.645,Z 733.66,A -85,B 0,C 180,E1 696.768,E2 696.768} C_VEL
LIN {X 0,Y 609.413,Z 733.66,A -85,B 0,C 180,E1 702.238,E2 702.238} C_VEL
LIN {X 0,Y 610.346,Z 765.038,A -85,B 0,C 180,E1 702.918,E2 702.918} C_VEL
LIN {X 0,Y 610.3,Z 792.759,A -85,B 0,C 180,E1 704.075,E2 704.075} C_VEL
LIN {X 0,Y 610.277,Z 817.804,A -85,B 0,C 180,E1 705.731,E2 705.731} C_VEL
LIN {X 0,Y 610.208,Z 839.182,A -85,B 0,C 180,E1 707.828,E2 707.828} C_VEL
LIN {X 0,Y 610.177,Z 854.32,A -85,B 0,C 180,E1 710.001,E2 710.001} C_VEL
LIN {X 0,Y 610.136,Z 865.646,A -85,B 0,C 180,E1 712.518,E2 712.518} C_VEL
LIN {X 0,Y 610.126,Z 871.629,A -85,B 0,C 180,E1 715.021,E2 715.021} C_VEL
LIN {X 0,Y 610.09,Z 872.959,A -85,B 0,C 180,E1 717.158,E2 717.158} C_VEL
LIN {X 0,Y 610.096,Z 869.551,A -85,B 0,C 180,E1 720.003,E2 720.003} C_VEL
LIN {X 0,Y 610.126,Z 861.39,A -85,B 0,C 180,E1 722.492,E2 722.492} C_VEL
LIN {X 0,Y 610.178,Z 847.531,A -85,B 0,C 180,E1 724.985,E2 724.985} C_VEL
LIN {X 0,Y 610.236,Z 829.572,A -85,B 0,C 180,E1 727.129,E2 727.129} C_VEL
LIN {X 0,Y 610.289,Z 806.485,A -85,B 0,C 180,E1 729.013,E2 729.013} C_VEL
LIN {X 0,Y 610.35,Z 779.734,A -85,B 0,C 180,E1 730.454,E2 730.454} C_VEL
LIN {X 0,Y 610.422,Z 751.032,A -85,B 0,C 180,E1 731.357,E2 731.357} C_VEL
LIN {X 0,Y 609.643,Z 733.66,A -85,B 0,C 180,E1 731.735,E2 731.735} C_VEL
LIN {X 0,Y 609.946,Z 733.66,A -85,B 0,C 180,E1 737.333,E2 737.333} C_VEL
LIN {X 0,Y 609.724,Z 733.66,A -85,B 0,C 180,E1 743.413,E2 743.413} C_VEL
LIN {X 0,Y 609.791,Z 733.66,A -85,B 0,C 180,E1 748.151,E2 748.151} C_VEL
LIN {X 0,Y 609.937,Z 733.66,A -85,B 0,C 180,E1 753.103,E2 753.103} C_VEL
LIN {X 0,Y 609.595,Z 733.66,A -85,B 0,C 180,E1 759.649,E2 759.649} C_VEL
LIN {X 0,Y 609.74,Z 733.66,A -85,B 0,C 180,E1 765.95,E2 765.95} C_VEL
LIN {X 0,Y 609.544,Z 733.66,A -85,B 0,C 180,E1 770.358,E2 770.358} C_VEL
LIN {X 0,Y 609.6,Z 733.66,A -85,B 0,C 180,E1 775.162,E2 775.162} C_VEL
LIN {X 0,Y 609.744,Z 733.66,A -85,B 0,C 180,E1 780.356,E2 780.356} C_VEL
LIN {X 0,Y 610.007,Z 733.66,A -85,B 0,C 180,E1 784.895,E2 784.895} C_VEL
LIN {X 0,Y 610.67,Z 779.456,A -85,B 0,C 180,E1 785.769,E2 785.769} C_VEL
LIN {X 0,Y 610.551,Z 816.363,A -85,B 0,C 180,E1 787.058,E2 787.058} C_VEL
LIN {X 0,Y 610.439,Z 850.057,A -85,B 0,C 180,E1 788.826,E2 788.826} C_VEL
LIN {X 0,Y 610.343,Z 880.861,A -85,B 0,C 180,E1 791.046,E2 791.046} C_VEL
LIN {X 0,Y 610.236,Z 909.301,A -85,B 0,C 180,E1 793.792,E2 793.792} C_VEL
LIN {X 0,Y 610.157,Z 932.004,A -85,B 0,C 180,E1 796.73,E2 796.73} C_VEL
LIN {X 0,Y 610.152,Z 950.439,A -85,B 0,C 180,E1 799.997,E2 799.997} C_VEL
LIN {X 0,Y 610.13,Z 963.963,A -85,B 0,C 180,E1 803.588,E2 803.588} C_VEL
LIN {X 0,Y 610.096,Z 971.22,A -85,B 0,C 180,E1 807.155,E2 807.155} C_VEL
LIN {X 0,Y 610.053,Z 972.996,A -85,B 0,C 180,E1 810,E2 810} C_VEL
LIN {X 0,Y 610.138,Z 970.09,A -85,B 0,C 180,E1 813.557,E2 813.557} C_VEL
LIN {X 0,Y 610.133,Z 961.459,A -85,B 0,C 180,E1 817.128,E2 817.128} C_VEL
LIN {X 0,Y 610.104,Z 948.254,A -85,B 0,C 180,E1 820.365,E2 820.365} C_VEL
LIN {X 0,Y 610.198,Z 928.971,A -85,B 0,C 180,E1 823.635,E2 823.635} C_VEL
LIN {X 0,Y 610.246,Z 905.071,A -85,B 0,C 180,E1 826.579,E2 826.579} C_VEL
LIN {X 0,Y 610.332,Z 876.612,A -85,B 0,C 180,E1 829.214,E2 829.214} C_VEL
LIN {X 0,Y 610.425,Z 843.825,A -85,B 0,C 180,E1 831.461,E2 831.461} C_VEL
LIN {X 0,Y 610.537,Z 809.545,A -85,B 0,C 180,E1 833.136,E2 833.136} C_VEL
LIN {X 0,Y 610.654,Z 773.278,A -85,B 0,C 180,E1 834.295,E2 834.295} C_VEL
LIN {X 0,Y 610.098,Z 733.66,A -85,B 0,C 180,E1 835.052,E2 835.052} C_VEL
LIN {X 0,Y 609.484,Z 733.66,A -85,B 0,C 180,E1 839.792,E2 839.792} C_VEL
LIN {X 0,Y 609.927,Z 733.66,A -85,B 0,C 180,E1 843.102,E2 843.102} C_VEL
LIN {X 0,Y 609.61,Z 733.66,A -85,B 0,C 180,E1 849.65,E2 849.65} C_VEL
LIN {X 0,Y 609.691,Z 733.66,A -85,B 0,C 180,E1 855.944,E2 855.944} C_VEL
LIN {X 0,Y 609.541,Z 733.66,A -85,B 0,C 180,E1 860.358,E2 860.358} C_VEL
LIN {X 0,Y 609.612,Z 733.66,A -85,B 0,C 180,E1 865.161,E2 865.161} C_VEL
LIN {X 0,Y 609.753,Z 733.66,A -85,B 0,C 180,E1 870.354,E2 870.354} C_VEL
LIN {X 0,Y 610.014,Z 733.66,A -85,B 0,C 180,E1 875.04,E2 875.04} C_VEL
LIN {X 0,Y 609.847,Z 733.66,A -85,B 0,C 180,E1 881.168,E2 881.168} C_VEL
LIN {X 0,Y 609.379,Z 733.66,A -85,B 0,C 180,E1 885.7,E2 885.7} C_VEL
LIN {X 0,Y 609.941,Z 733.66,A -85,B 0,C 180,E1 889.991,E2 889.991} C_VEL
LIN {X 0,Y 609.948,Z 733.66,A -85,B 0,C 180,E1 894.603,E2 894.603} C_VEL
LIN {X 0,Y 605.702,Z 733.66,A -85,B 0,C 180,E1 896.199,E2 896.199} C_VEL
LIN {X 0,Y 601.92,Z 733.66,A -85,B 0,C 180,E1 897.817,E2 897.817} C_VEL
LIN {X 0,Y 602.002,Z 733.66,A -85,B 0,C 180,E1 902.88,E2 902.88} C_VEL
LIN {X 0,Y 602.018,Z 733.66,A -85,B 0,C 180,E1 908.675,E2 908.675} C_VEL
LIN {X 0,Y 602.106,Z 733.66,A -85,B 0,C 180,E1 913.076,E2 913.076} C_VEL
LIN {X 0,Y 602.075,Z 733.66,A -85,B 0,C 180,E1 917.56,E2 917.56} C_VEL
LIN {X 0,Y 601.766,Z 733.66,A -85,B 0,C 180,E1 923.734,E2 923.734} C_VEL
LIN {X 0,Y 601.785,Z 733.66,A -85,B 0,C 180,E1 928.552,E2 928.552} C_VEL
LIN {X 0,Y 601.83,Z 733.66,A -85,B 0,C 180,E1 933.878,E2 933.878} C_VEL
LIN {X 0,Y 601.758,Z 733.66,A -85,B 0,C 180,E1 938.972,E2 938.972} C_VEL
LIN {X 0,Y 601.739,Z 733.66,A -85,B 0,C 180,E1 945.208,E2 945.208} C_VEL
LIN {X 0,Y 601.737,Z 733.66,A -85,B 0,C 180,E1 951.254,E2 951.254} C_VEL
LIN {X 0,Y 601.543,Z 733.66,A -85,B 0,C 180,E1 956.376,E2 956.376} C_VEL
LIN {X 0,Y 601.703,Z 733.66,A -85,B 0,C 180,E1 961.717,E2 961.717} C_VEL
LIN {X 0,Y 601.803,Z 733.66,A -85,B 0,C 180,E1 963.953,E2 963.953} C_VEL
LIN {X 0,Y 603.43,Z 750.904,A -85,B 0,C 180,E1 964.255,E2 964.255} C_VEL
LIN {X 0,Y 603.417,Z 819.07,A -85,B 0,C 180,E1 965.246,E2 965.246} C_VEL
LIN {X 0,Y 603.293,Z 855.864,A -85,B 0,C 180,E1 966.373,E2 966.373} C_VEL
LIN {X 0,Y 603.022,Z 890.418,A -85,B 0,C 180,E1 968.02,E2 968.02} C_VEL
LIN {X 0,Y 602.753,Z 923.4,A -85,B 0,C 180,E1 970.232,E2 970.232} C_VEL
LIN {X 0,Y 602.475,Z 952.3,A -85,B 0,C 180,E1 972.859,E2 972.859} C_VEL
LIN {X 0,Y 602.313,Z 976.641,A -85,B 0,C 180,E1 975.812,E2 975.812} C_VEL
LIN {X 0,Y 602.191,Z 995.809,A -85,B 0,C 180,E1 978.958,E2 978.958} C_VEL
LIN {X 0,Y 602.137,Z 1010.458,A -85,B 0,C 180,E1 982.414,E2 982.414} C_VEL
LIN {X 0,Y 602.104,Z 1018.972,A -85,B 0,C 180,E1 985.673,E2 985.673} C_VEL
LIN {X 0,Y 602.118,Z 1022.509,A -85,B 0,C 180,E1 988.559,E2 988.559} C_VEL
LIN {X 0,Y 602.212,Z 1022.509,A -85,B 0,C 180,E1 991.44,E2 991.44} C_VEL
LIN {X 0,Y 602.177,Z 1017.453,A -85,B 0,C 180,E1 995.049,E2 995.049} C_VEL
LIN {X 0,Y 602.192,Z 1006.499,A -85,B 0,C 180,E1 998.676,E2 998.676} C_VEL
LIN {X 0,Y 602.249,Z 989.708,A -85,B 0,C 180,E1 1002.155,E2 1002.155} C_VEL
LIN {X 0,Y 602.381,Z 968.267,A -85,B 0,C 180,E1 1005.303,E2 1005.303} C_VEL
LIN {X 0,Y 602.598,Z 941.58,A -85,B 0,C 180,E1 1008.21,E2 1008.21} C_VEL
LIN {X 0,Y 602.839,Z 911.345,A -85,B 0,C 180,E1 1010.658,E2 1010.658} C_VEL
LIN {X 0,Y 603.156,Z 877.997,A -85,B 0,C 180,E1 1012.643,E2 1012.643} C_VEL
LIN {X 0,Y 603.392,Z 842.296,A -85,B 0,C 180,E1 1014.113,E2 1014.113} C_VEL
LIN {X 0,Y 603.545,Z 806.699,A -85,B 0,C 180,E1 1014.996,E2 1014.996} C_VEL
LIN {X 0,Y 602.633,Z 738.705,A -85,B 0,C 180,E1 1015.94,E2 1015.94} C_VEL
LIN {X 0,Y 601.846,Z 733.66,A -85,B 0,C 180,E1 1016.121,E2 1016.121} C_VEL
LIN {X 0,Y 601.639,Z 733.66,A -85,B 0,C 180,E1 1021.903,E2 1021.903} C_VEL
LIN {X 0,Y 601.736,Z 733.66,A -85,B 0,C 180,E1 1027.149,E2 1027.149} C_VEL
LIN {X 0,Y 601.777,Z 733.66,A -85,B 0,C 180,E1 1033.151,E2 1033.151} C_VEL
LIN {X 0,Y 601.568,Z 733.66,A -85,B 0,C 180,E1 1039.133,E2 1039.133} C_VEL
LIN {X 0,Y 601.493,Z 733.66,A -85,B 0,C 180,E1 1043.659,E2 1043.659} C_VEL
LIN {X 0,Y 601.812,Z 733.66,A -85,B 0,C 180,E1 1048.113,E2 1048.113} C_VEL
LIN {X 0,Y 601.64,Z 733.66,A -85,B 0,C 180,E1 1053.07,E2 1053.07} C_VEL
LIN {X 0,Y 601.647,Z 733.66,A -85,B 0,C 180,E1 1058.612,E2 1058.612} C_VEL
LIN {X 0,Y 601.75,Z 734.288,A -85,B 0,C 180,E1 1062.067,E2 1062.067} C_VEL
LIN {X 0,Y 602.695,Z 763.592,A -85,B 0,C 180,E1 1062.691,E2 1062.691} C_VEL
LIN {X 0,Y 602.587,Z 792.247,A -85,B 0,C 180,E1 1063.879,E2 1063.879} C_VEL
LIN {X 0,Y 602.474,Z 817.288,A -85,B 0,C 180,E1 1065.542,E2 1065.542} C_VEL
LIN {X 0,Y 602.389,Z 838.857,A -85,B 0,C 180,E1 1067.668,E2 1067.668} C_VEL
LIN {X 0,Y 602.29,Z 854.094,A -85,B 0,C 180,E1 1069.869,E2 1069.869} C_VEL
LIN {X 0,Y 602.229,Z 865.513,A -85,B 0,C 180,E1 1072.419,E2 1072.419} C_VEL
LIN {X 0,Y 602.221,Z 871.564,A -85,B 0,C 180,E1 1074.955,E2 1074.955} C_VEL
LIN {X 0,Y 602.188,Z 872.97,A -85,B 0,C 180,E1 1077.121,E2 1077.121} C_VEL
LIN {X 0,Y 602.197,Z 869.64,A -85,B 0,C 180,E1 1080.003,E2 1080.003} C_VEL
LIN {X 0,Y 602.238,Z 861.556,A -85,B 0,C 180,E1 1082.525,E2 1082.525} C_VEL
LIN {X 0,Y 602.316,Z 847.8,A -85,B 0,C 180,E1 1085.051,E2 1085.051} C_VEL
LIN {X 0,Y 602.404,Z 829.967,A -85,B 0,C 180,E1 1087.222,E2 1087.222} C_VEL
LIN {X 0,Y 602.509,Z 807.099,A -85,B 0,C 180,E1 1089.13,E2 1089.13} C_VEL
LIN {X 0,Y 602.633,Z 780.782,A -85,B 0,C 180,E1 1090.585,E2 1090.585} C_VEL
LIN {X 0,Y 602.761,Z 751.662,A -85,B 0,C 180,E1 1091.529,E2 1091.529} C_VEL
LIN {X 0,Y 601.878,Z 733.66,A -85,B 0,C 180,E1 1091.864,E2 1091.864} C_VEL
LIN {X 0,Y 602.009,Z 733.66,A -85,B 0,C 180,E1 1097.569,E2 1097.569} C_VEL
LIN {X 0,Y 601.747,Z 733.66,A -85,B 0,C 180,E1 1103.742,E2 1103.742} C_VEL
LIN {X 0,Y 601.777,Z 733.66,A -85,B 0,C 180,E1 1108.56,E2 1108.56} C_VEL
LIN {X 0,Y 601.828,Z 733.66,A -85,B 0,C 180,E1 1113.879,E2 1113.879} C_VEL
LIN {X 0,Y 601.767,Z 733.66,A -85,B 0,C 180,E1 1118.979,E2 1118.979} C_VEL
LIN {X 0,Y 601.743,Z 733.66,A -85,B 0,C 180,E1 1125.209,E2 1125.209} C_VEL
LIN {X 0,Y 601.706,Z 733.66,A -85,B 0,C 180,E1 1131.018,E2 1131.018} C_VEL
LIN {X 0,Y 601.555,Z 733.66,A -85,B 0,C 180,E1 1136.161,E2 1136.161} C_VEL
LIN {X 0,Y 601.601,Z 733.66,A -85,B 0,C 180,E1 1141.433,E2 1141.433} C_VEL
LIN {X 0,Y 602.112,Z 733.66,A -85,B 0,C 180,E1 1144.569,E2 1144.569} C_VEL
LIN {X 0,Y 603.378,Z 749.32,A -85,B 0,C 180,E1 1144.839,E2 1144.839} C_VEL
LIN {X 0,Y 603.35,Z 787.341,A -85,B 0,C 180,E1 1145.688,E2 1145.688} C_VEL
LIN {X 0,Y 603.162,Z 823.522,A -85,B 0,C 180,E1 1147.091,E2 1147.091} C_VEL
LIN {X 0,Y 602.874,Z 857.945,A -85,B 0,C 180,E1 1149.061,E2 1149.061} C_VEL
LIN {X 0,Y 602.641,Z 888.937,A -85,B 0,C 180,E1 1151.507,E2 1151.507} C_VEL
LIN {X 0,Y 602.424,Z 915.681,A -85,B 0,C 180,E1 1154.325,E2 1154.325} C_VEL
LIN {X 0,Y 602.287,Z 937.793,A -85,B 0,C 180,E1 1157.478,E2 1157.478} C_VEL
LIN {X 0,Y 602.266,Z 953.662,A -85,B 0,C 180,E1 1160.595,E2 1160.595} C_VEL
LIN {X 0,Y 602.233,Z 964.533,A -85,B 0,C 180,E1 1163.719,E2 1163.719} C_VEL
LIN {X 0,Y 602.194,Z 971.22,A -85,B 0,C 180,E1 1167.118,E2 1167.118} C_VEL
LIN {X 0,Y 602.153,Z 972.996,A -85,B 0,C 180,E1 1170,E2 1170} C_VEL
LIN {X 0,Y 602.246,Z 970.091,A -85,B 0,C 180,E1 1173.604,E2 1173.604} C_VEL
LIN {X 0,Y 602.232,Z 961.462,A -85,B 0,C 180,E1 1177.222,E2 1177.222} C_VEL
LIN {X 0,Y 602.28,Z 947.18,A -85,B 0,C 180,E1 1180.728,E2 1180.728} C_VEL
LIN {X 0,Y 602.374,Z 927.652,A -85,B 0,C 180,E1 1184.001,E2 1184.001} C_VEL
LIN {X 0,Y 602.509,Z 903.418,A -85,B 0,C 180,E1 1186.976,E2 1186.976} C_VEL
LIN {X 0,Y 602.749,Z 874.117,A -85,B 0,C 180,E1 1189.668,E2 1189.668} C_VEL
LIN {X 0,Y 602.959,Z 842.463,A -85,B 0,C 180,E1 1191.819,E2 1191.819} C_VEL
LIN {X 0,Y 603.267,Z 808.2,A -85,B 0,C 180,E1 1193.487,E2 1193.487} C_VEL
LIN {X 0,Y 603.487,Z 770.722,A -85,B 0,C 180,E1 1194.667,E2 1194.667} C_VEL
LIN {X 0,Y 602.748,Z 736.707,A -85,B 0,C 180,E1 1195.268,E2 1195.268} C_VEL
LIN {X 0,Y 602.131,Z 733.66,A -85,B 0,C 180,E1 1195.407,E2 1195.407} C_VEL
LIN {X 0,Y 601.582,Z 733.66,A -85,B 0,C 180,E1 1201.159,E2 1201.159} C_VEL
LIN {X 0,Y 601.594,Z 733.66,A -85,B 0,C 180,E1 1205.371,E2 1205.371} C_VEL
LIN {X 0,Y 601.774,Z 733.66,A -85,B 0,C 180,E1 1208.978,E2 1208.978} C_VEL
LIN {X 0,Y 601.702,Z 733.66,A -85,B 0,C 180,E1 1215.203,E2 1215.203} C_VEL
LIN {X 0,Y 601.664,Z 733.66,A -85,B 0,C 180,E1 1221.013,E2 1221.013} C_VEL
LIN {X 0,Y 601.546,Z 733.66,A -85,B 0,C 180,E1 1226.162,E2 1226.162} C_VEL
LIN {X 0,Y 601.652,Z 733.66,A -85,B 0,C 180,E1 1231.434,E2 1231.434} C_VEL
LIN {X 0,Y 601.752,Z 733.66,A -85,B 0,C 180,E1 1236.258,E2 1236.258} C_VEL
LIN {X 0,Y 601.975,Z 733.66,A -85,B 0,C 180,E1 1240.912,E2 1240.912} C_VEL
LIN {X 0,Y 601.54,Z 733.66,A -85,B 0,C 180,E1 1245.419,E2 1245.419} C_VEL
LIN {X 0,Y 601.998,Z 733.66,A -85,B 0,C 180,E1 1249.857,E2 1249.857} C_VEL
LIN {X 0,Y 602.029,Z 733.66,A -85,B 0,C 180,E1 1254.58,E2 1254.58} C_VEL
LIN {X 0,Y 601.92,Z 733.66,A -85,B 0,C 180,E1 1257.817,E2 1257.817} C_VEL
LIN {X 0,Y 599.482,Z 733.66,A -85,B 0,C 180,E1 1259.046,E2 1259.046} C_VEL
LIN {X 0,Y 593.95,Z 733.66,A -85,B 0,C 180,E1 1260.885,E2 1260.885} C_VEL
LIN {X 0,Y 593.847,Z 733.66,A -85,B 0,C 180,E1 1261.097,E2 1261.097} C_VEL
LIN {X 0,Y 593.855,Z 733.66,A -85,B 0,C 180,E1 1266.094,E2 1266.094} C_VEL
LIN {X 0,Y 593.843,Z 733.66,A -85,B 0,C 180,E1 1270.277,E2 1270.277} C_VEL
LIN {X 0,Y 593.812,Z 733.66,A -85,B 0,C 180,E1 1274.768,E2 1274.768} C_VEL
LIN {X 0,Y 593.913,Z 733.66,A -85,B 0,C 180,E1 1279.393,E2 1279.393} C_VEL
LIN {X 0,Y 593.84,Z 733.66,A -85,B 0,C 180,E1 1284.071,E2 1284.071} C_VEL
LIN {X 0,Y 593.779,Z 733.66,A -85,B 0,C 180,E1 1288.973,E2 1288.973} C_VEL
LIN {X 0,Y 593.888,Z 733.66,A -85,B 0,C 180,E1 1294.111,E2 1294.111} C_VEL
LIN {X 0,Y 593.681,Z 733.66,A -85,B 0,C 180,E1 1300.083,E2 1300.083} C_VEL
LIN {X 0,Y 593.805,Z 733.66,A -85,B 0,C 180,E1 1305.549,E2 1305.549} C_VEL
LIN {X 0,Y 593.74,Z 733.66,A -85,B 0,C 180,E1 1310.392,E2 1310.392} C_VEL
LIN {X 0,Y 593.677,Z 733.66,A -85,B 0,C 180,E1 1315.869,E2 1315.869} C_VEL
LIN {X 0,Y 593.8,Z 733.66,A -85,B 0,C 180,E1 1321.022,E2 1321.022} C_VEL
LIN {X 0,Y 593.948,Z 733.66,A -85,B 0,C 180,E1 1323.58,E2 1323.58} C_VEL
LIN {X 0,Y 596.303,Z 748.416,A -85,B 0,C 180,E1 1323.892,E2 1323.892} C_VEL
LIN {X 0,Y 596.244,Z 818.995,A -85,B 0,C 180,E1 1324.926,E2 1324.926} C_VEL
LIN {X 0,Y 595.979,Z 856.685,A -85,B 0,C 180,E1 1326.099,E2 1326.099} C_VEL
LIN {X 0,Y 595.575,Z 891.402,A -85,B 0,C 180,E1 1327.788,E2 1327.788} C_VEL
LIN {X 0,Y 595.182,Z 924.082,A -85,B 0,C 180,E1 1330.022,E2 1330.022} C_VEL
LIN {X 0,Y 594.747,Z 953.576,A -85,B 0,C 180,E1 1332.768,E2 1332.768} C_VEL
LIN {X 0,Y 594.494,Z 978.59,A -85,B 0,C 180,E1 1335.896,E2 1335.896} C_VEL
LIN {X 0,Y 594.294,Z 997.698,A -85,B 0,C 180,E1 1339.19,E2 1339.19} C_VEL
LIN {X 0,Y 594.258,Z 1011.606,A -85,B 0,C 180,E1 1342.681,E2 1342.681} C_VEL
LIN {X 0,Y 594.214,Z 1020.171,A -85,B 0,C 180,E1 1346.347,E2 1346.347} C_VEL
LIN {X 0,Y 594.195,Z 1023,A -85,B 0,C 180,E1 1350,E2 1350} C_VEL
LIN {X 0,Y 594.284,Z 1020.172,A -85,B 0,C 180,E1 1353.652,E2 1353.652} C_VEL
LIN {X 0,Y 594.305,Z 1011.606,A -85,B 0,C 180,E1 1357.318,E2 1357.318} C_VEL
LIN {X 0,Y 594.389,Z 997.599,A -85,B 0,C 180,E1 1360.83,E2 1360.83} C_VEL
LIN {X 0,Y 594.574,Z 977.254,A -85,B 0,C 180,E1 1364.29,E2 1364.29} C_VEL
LIN {X 0,Y 594.829,Z 952.14,A -85,B 0,C 180,E1 1367.386,E2 1367.386} C_VEL
LIN {X 0,Y 595.157,Z 922.064,A -85,B 0,C 180,E1 1370.136,E2 1370.136} C_VEL
LIN {X 0,Y 595.588,Z 889.638,A -85,B 0,C 180,E1 1372.315,E2 1372.315} C_VEL
LIN {X 0,Y 595.948,Z 853.45,A -85,B 0,C 180,E1 1374.033,E2 1374.033} C_VEL
LIN {X 0,Y 596.224,Z 817.081,A -85,B 0,C 180,E1 1375.117,E2 1375.117} C_VEL
LIN {X 0,Y 595.594,Z 740.273,A -85,B 0,C 180,E1 1376.249,E2 1376.249} C_VEL
LIN {X 0,Y 593.93,Z 733.66,A -85,B 0,C 180,E1 1376.471,E2 1376.471} C_VEL
LIN {X 0,Y 593.875,Z 733.66,A -85,B 0,C 180,E1 1380.657,E2 1380.657} C_VEL
LIN {X 0,Y 593.842,Z 733.66,A -85,B 0,C 180,E1 1385.903,E2 1385.903} C_VEL
LIN {X 0,Y 593.799,Z 733.66,A -85,B 0,C 180,E1 1391.526,E2 1391.526} C_VEL
LIN {X 0,Y 593.715,Z 733.66,A -85,B 0,C 180,E1 1396.492,E2 1396.492} C_VEL
LIN {X 0,Y 593.704,Z 733.66,A -85,B 0,C 180,E1 1402.268,E2 1402.268} C_VEL
LIN {X 0,Y 593.884,Z 733.66,A -85,B 0,C 180,E1 1407.636,E2 1407.636} C_VEL
LIN {X 0,Y 593.727,Z 733.66,A -85,B 0,C 180,E1 1413.195,E2 1413.195} C_VEL
LIN {X 0,Y 593.758,Z 733.66,A -85,B 0,C 180,E1 1417.516,E2 1417.516} C_VEL
LIN {X 0,Y 593.93,Z 733.66,A -85,B 0,C 180,E1 1421.855,E2 1421.855} C_VEL
LIN {X 0,Y 595.044,Z 762.715,A -85,B 0,C 180,E1 1422.477,E2 1422.477} C_VEL
LIN {X 0,Y 594.867,Z 791.68,A -85,B 0,C 180,E1 1423.674,E2 1423.674} C_VEL
LIN {X 0,Y 594.699,Z 816.738,A -85,B 0,C 180,E1 1425.346,E2 1425.346} C_VEL
LIN {X 0,Y 594.515,Z 838.513,A -85,B 0,C 180,E1 1427.502,E2 1427.502} C_VEL
LIN {X 0,Y 594.424,Z 853.865,A -85,B 0,C 180,E1 1429.733,E2 1429.733} C_VEL
LIN {X 0,Y 594.338,Z 865.365,A -85,B 0,C 180,E1 1432.318,E2 1432.318} C_VEL
LIN {X 0,Y 594.351,Z 871.492,A -85,B 0,C 180,E1 1434.888,E2 1434.888} C_VEL
LIN {X 0,Y 594.285,Z 872.978,A -85,B 0,C 180,E1 1437.083,E2 1437.083} C_VEL
LIN {X 0,Y 594.299,Z 869.729,A -85,B 0,C 180,E1 1440.003,E2 1440.003} C_VEL
LIN {X 0,Y 594.343,Z 861.722,A -85,B 0,C 180,E1 1442.558,E2 1442.558} C_VEL
LIN {X 0,Y 594.449,Z 848.068,A -85,B 0,C 180,E1 1445.118,E2 1445.118} C_VEL
LIN {X 0,Y 594.58,Z 830.36,A -85,B 0,C 180,E1 1447.318,E2 1447.318} C_VEL
LIN {X 0,Y 594.735,Z 806.351,A -85,B 0,C 180,E1 1449.343,E2 1449.343} C_VEL
LIN {X 0,Y 594.957,Z 780.371,A -85,B 0,C 180,E1 1450.783,E2 1450.783} C_VEL
LIN {X 0,Y 595.129,Z 752.655,A -85,B 0,C 180,E1 1451.696,E2 1451.696} C_VEL
LIN {X 0,Y 594.181,Z 733.66,A -85,B 0,C 180,E1 1452.092,E2 1452.092} C_VEL
LIN {X 0,Y 594.053,Z 733.66,A -85,B 0,C 180,E1 1457.812,E2 1457.812} C_VEL
LIN {X 0,Y 593.81,Z 733.66,A -85,B 0,C 180,E1 1464.079,E2 1464.079} C_VEL
LIN {X 0,Y 593.77,Z 733.66,A -85,B 0,C 180,E1 1468.981,E2 1468.981} C_VEL
LIN {X 0,Y 593.886,Z 733.66,A -85,B 0,C 180,E1 1474.119,E2 1474.119} C_VEL
LIN {X 0,Y 593.684,Z 733.66,A -85,B 0,C 180,E1 1480.084,E2 1480.084} C_VEL
LIN {X 0,Y 593.811,Z 733.66,A -85,B 0,C 180,E1 1485.558,E2 1485.558} C_VEL
LIN {X 0,Y 593.74,Z 733.66,A -85,B 0,C 180,E1 1490.393,E2 1490.393} C_VEL
LIN {X 0,Y 593.666,Z 733.66,A -85,B 0,C 180,E1 1495.869,E2 1495.869} C_VEL
LIN {X 0,Y 593.703,Z 733.66,A -85,B 0,C 180,E1 1501.017,E2 1501.017} C_VEL
LIN {X 0,Y 594.072,Z 733.66,A -85,B 0,C 180,E1 1504.184,E2 1504.184} C_VEL
LIN {X 0,Y 596.251,Z 742.762,A -85,B 0,C 180,E1 1504.425,E2 1504.425} C_VEL
LIN {X 0,Y 596.235,Z 780.737,A -85,B 0,C 180,E1 1505.18,E2 1505.18} C_VEL
LIN {X 0,Y 595.887,Z 816.966,A -85,B 0,C 180,E1 1506.489,E2 1506.489} C_VEL
LIN {X 0,Y 595.442,Z 850.616,A -85,B 0,C 180,E1 1508.303,E2 1508.303} C_VEL
LIN {X 0,Y 595.077,Z 882.548,A -85,B 0,C 180,E1 1510.685,E2 1510.685} C_VEL
LIN {X 0,Y 594.72,Z 910.206,A -85,B 0,C 180,E1 1513.465,E2 1513.465} C_VEL
LIN {X 0,Y 594.525,Z 933.35,A -85,B 0,C 180,E1 1516.584,E2 1516.584} C_VEL
LIN {X 0,Y 594.407,Z 952.121,A -85,B 0,C 180,E1 1520.1,E2 1520.1} C_VEL
LIN {X 0,Y 594.346,Z 964.115,A -85,B 0,C 180,E1 1523.476,E2 1523.476} C_VEL
LIN {X 0,Y 594.293,Z 971.219,A -85,B 0,C 180,E1 1527.079,E2 1527.079} C_VEL
LIN {X 0,Y 594.253,Z 972.996,A -85,B 0,C 180,E1 1530,E2 1530} C_VEL
LIN {X 0,Y 594.348,Z 970.092,A -85,B 0,C 180,E1 1533.652,E2 1533.652} C_VEL
LIN {X 0,Y 594.353,Z 961.465,A -85,B 0,C 180,E1 1537.318,E2 1537.318} C_VEL
LIN {X 0,Y 594.402,Z 947.507,A -85,B 0,C 180,E1 1540.803,E2 1540.803} C_VEL
LIN {X 0,Y 594.576,Z 927.085,A -85,B 0,C 180,E1 1544.269,E2 1544.269} C_VEL
LIN {X 0,Y 594.832,Z 901.933,A -85,B 0,C 180,E1 1547.364,E2 1547.364} C_VEL
LIN {X 0,Y 595.194,Z 872.634,A -85,B 0,C 180,E1 1550.044,E2 1550.044} C_VEL
LIN {X 0,Y 595.59,Z 840.832,A -85,B 0,C 180,E1 1552.199,E2 1552.199} C_VEL
LIN {X 0,Y 596.012,Z 805.629,A -85,B 0,C 180,E1 1553.898,E2 1553.898} C_VEL
LIN {X 0,Y 596.305,Z 769.832,A -85,B 0,C 180,E1 1555.008,E2 1555.008} C_VEL
LIN {X 0,Y 595.497,Z 738.087,A -85,B 0,C 180,E1 1555.581,E2 1555.581} C_VEL
LIN {X 0,Y 594.2,Z 733.66,A -85,B 0,C 180,E1 1555.745,E2 1555.745} C_VEL
LIN {X 0,Y 593.799,Z 733.66,A -85,B 0,C 180,E1 1562.376,E2 1562.376} C_VEL
LIN {X 0,Y 593.704,Z 733.66,A -85,B 0,C 180,E1 1567.759,E2 1567.759} C_VEL
LIN {X 0,Y 593.691,Z 733.66,A -85,B 0,C 180,E1 1573.518,E2 1573.518} C_VEL
LIN {X 0,Y 593.788,Z 733.66,A -85,B 0,C 180,E1 1578.472,E2 1578.472} C_VEL
LIN {X 0,Y 593.826,Z 733.66,A -85,B 0,C 180,E1 1584.094,E2 1584.094} C_VEL
LIN {X 0,Y 593.827,Z 733.66,A -85,B 0,C 180,E1 1590.101,E2 1590.101} C_VEL
LIN {X 0,Y 593.919,Z 733.66,A -85,B 0,C 180,E1 1595.925,E2 1595.925} C_VEL
LIN {X 0,Y 594.049,Z 733.66,A -85,B 0,C 180,E1 1600.648,E2 1600.648} C_VEL
LIN {X 0,Y 593.698,Z 733.66,A -85,B 0,C 180,E1 1605.222,E2 1605.222} C_VEL
LIN {X 0,Y 594.059,Z 733.66,A -85,B 0,C 180,E1 1609.72,E2 1609.72} C_VEL
LIN {X 0,Y 594.221,Z 733.66,A -85,B 0,C 180,E1 1614.147,E2 1614.147} C_VEL
LIN {X 0,Y 593.995,Z 733.66,A -85,B 0,C 180,E1 1619.997,E2 1619.997} C_VEL
LIN {X 0,Y 593.847,Z 733.66,A -85,B 0,C 180,E1 1621.097,E2 1621.097} C_VEL
LIN {X 0,Y 589.949,Z 733.66,A -85,B 0,C 180,E1 1622.751,E2 1622.751} C_VEL
LIN {X 0,Y 586.144,Z 733.66,A -85,B 0,C 180,E1 1624.427,E2 1624.427} C_VEL
LIN {X 0,Y 586.16,Z 733.66,A -85,B 0,C 180,E1 1628.912,E2 1628.912} C_VEL
LIN {X 0,Y 586.189,Z 733.66,A -85,B 0,C 180,E1 1633.438,E2 1633.438} C_VEL
LIN {X 0,Y 586.158,Z 733.66,A -85,B 0,C 180,E1 1638.053,E2 1638.053} C_VEL
LIN {X 0,Y 586.017,Z 733.66,A -85,B 0,C 180,E1 1642.797,E2 1642.797} C_VEL
LIN {X 0,Y 585.867,Z 733.66,A -85,B 0,C 180,E1 1648.516,E2 1648.516} C_VEL
LIN {X 0,Y 585.873,Z 733.66,A -85,B 0,C 180,E1 1654.643,E2 1654.643} C_VEL
LIN {X 0,Y 585.787,Z 733.66,A -85,B 0,C 180,E1 1660.247,E2 1660.247} C_VEL
LIN {X 0,Y 585.923,Z 733.66,A -85,B 0,C 180,E1 1666.34,E2 1666.34} C_VEL
LIN {X 0,Y 585.848,Z 733.66,A -85,B 0,C 180,E1 1671.664,E2 1671.664} C_VEL
LIN {X 0,Y 585.747,Z 733.66,A -85,B 0,C 180,E1 1677.123,E2 1677.123} C_VEL
LIN {X 0,Y 586.059,Z 733.66,A -85,B 0,C 180,E1 1683.164,E2 1683.164} C_VEL
LIN {X 0,Y 589.199,Z 746.432,A -85,B 0,C 180,E1 1683.526,E2 1683.526} C_VEL
LIN {X 0,Y 589.095,Z 819.119,A -85,B 0,C 180,E1 1684.604,E2 1684.604} C_VEL
LIN {X 0,Y 588.707,Z 856.04,A -85,B 0,C 180,E1 1685.757,E2 1685.757} C_VEL
LIN {X 0,Y 588.135,Z 891.497,A -85,B 0,C 180,E1 1687.497,E2 1687.497} C_VEL
LIN {X 0,Y 587.595,Z 923.568,A -85,B 0,C 180,E1 1689.712,E2 1689.712} C_VEL
LIN {X 0,Y 587.066,Z 953.027,A -85,B 0,C 180,E1 1692.474,E2 1692.474} C_VEL
LIN {X 0,Y 586.707,Z 978.117,A -85,B 0,C 180,E1 1695.636,E2 1695.636} C_VEL
LIN {X 0,Y 586.485,Z 996.459,A -85,B 0,C 180,E1 1698.786,E2 1698.786} C_VEL
LIN {X 0,Y 586.382,Z 1010.451,A -85,B 0,C 180,E1 1702.209,E2 1702.209} C_VEL
LIN {X 0,Y 586.308,Z 1018.974,A -85,B 0,C 180,E1 1705.556,E2 1705.556} C_VEL
LIN {X 0,Y 586.32,Z 1022.514,A -85,B 0,C 180,E1 1708.52,E2 1708.52} C_VEL
LIN {X 0,Y 586.403,Z 1022.514,A -85,B 0,C 180,E1 1711.479,E2 1711.479} C_VEL
LIN {X 0,Y 586.406,Z 1017.457,A -85,B 0,C 180,E1 1715.185,E2 1715.185} C_VEL
LIN {X 0,Y 586.411,Z 1006.491,A -85,B 0,C 180,E1 1718.912,E2 1718.912} C_VEL
LIN {X 0,Y 586.567,Z 990.794,A -85,B 0,C 180,E1 1722.295,E2 1722.295} C_VEL
LIN {X 0,Y 586.808,Z 969.744,A -85,B 0,C 180,E1 1725.527,E2 1725.527} C_VEL
LIN {X 0,Y 587.235,Z 944.498,A -85,B 0,C 180,E1 1728.412,E2 1728.412} C_VEL
LIN {X 0,Y 587.756,Z 914.368,A -85,B 0,C 180,E1 1730.996,E2 1730.996} C_VEL
LIN {X 0,Y 588.363,Z 880.895,A -85,B 0,C 180,E1 1733.092,E2 1733.092} C_VEL
LIN {X 0,Y 588.837,Z 846.547,A -85,B 0,C 180,E1 1734.597,E2 1734.597} C_VEL
LIN {X 0,Y 589.222,Z 810.651,A -85,B 0,C 180,E1 1735.571,E2 1735.571} C_VEL
LIN {X 0,Y 588.628,Z 742.123,A -85,B 0,C 180,E1 1736.559,E2 1736.559} C_VEL
LIN {X 0,Y 586.076,Z 733.66,A -85,B 0,C 180,E1 1736.851,E2 1736.851} C_VEL
LIN {X 0,Y 585.744,Z 733.66,A -85,B 0,C 180,E1 1742.876,E2 1742.876} C_VEL
LIN {X 0,Y 585.814,Z 733.66,A -85,B 0,C 180,E1 1748.338,E2 1748.338} C_VEL
LIN {X 0,Y 585.91,Z 733.66,A -85,B 0,C 180,E1 1754.245,E2 1754.245} C_VEL
LIN {X 0,Y 585.786,Z 733.66,A -85,B 0,C 180,E1 1759.753,E2 1759.753} C_VEL
LIN {X 0,Y 585.968,Z 733.66,A -85,B 0,C 180,E1 1765.776,E2 1765.776} C_VEL
LIN {X 0,Y 585.85,Z 733.66,A -85,B 0,C 180,E1 1771.487,E2 1771.487} C_VEL
LIN {X 0,Y 585.871,Z 733.66,A -85,B 0,C 180,E1 1777.196,E2 1777.196} C_VEL
LIN {X 0,Y 586.053,Z 733.66,A -85,B 0,C 180,E1 1781.641,E2 1781.641} C_VEL
LIN {X 0,Y 587.405,Z 761.729,A -85,B 0,C 180,E1 1782.255,E2 1782.255} C_VEL
LIN {X 0,Y 587.197,Z 789.823,A -85,B 0,C 180,E1 1783.402,E2 1783.402} C_VEL
LIN {X 0,Y 586.926,Z 815.104,A -85,B 0,C 180,E1 1785.055,E2 1785.055} C_VEL
LIN {X 0,Y 586.691,Z 836.528,A -85,B 0,C 180,E1 1787.143,E2 1787.143} C_VEL
LIN {X 0,Y 586.538,Z 853.63,A -85,B 0,C 180,E1 1789.594,E2 1789.594} C_VEL
LIN {X 0,Y 586.458,Z 865.217,A -85,B 0,C 180,E1 1792.214,E2 1792.214} C_VEL
LIN {X 0,Y 586.466,Z 871.42,A -85,B 0,C 180,E1 1794.819,E2 1794.819} C_VEL
LIN {X 0,Y 586.387,Z 872.969,A -85,B 0,C 180,E1 1797.043,E2 1797.043} C_VEL
LIN {X 0,Y 586.4,Z 869.818,A -85,B 0,C 180,E1 1800.003,E2 1800.003} C_VEL
LIN {X 0,Y 586.46,Z 861.888,A -85,B 0,C 180,E1 1802.593,E2 1802.593} C_VEL
LIN {X 0,Y 586.576,Z 848.338,A -85,B 0,C 180,E1 1805.186,E2 1805.186} C_VEL
LIN {X 0,Y 586.767,Z 830.752,A -85,B 0,C 180,E1 1807.416,E2 1807.416} C_VEL
LIN {X 0,Y 586.962,Z 806.953,A -85,B 0,C 180,E1 1809.468,E2 1809.468} C_VEL
LIN {X 0,Y 587.26,Z 781.24,A -85,B 0,C 180,E1 1810.929,E2 1810.929} C_VEL
LIN {X 0,Y 587.494,Z 752.241,A -85,B 0,C 180,E1 1811.901,E2 1811.901} C_VEL
LIN {X 0,Y 586.294,Z 733.66,A -85,B 0,C 180,E1 1812.269,E2 1812.269} C_VEL
LIN {X 0,Y 586.098,Z 733.66,A -85,B 0,C 180,E1 1818.062,E2 1818.062} C_VEL
LIN {X 0,Y 586,Z 733.66,A -85,B 0,C 180,E1 1822.805,E2 1822.805} C_VEL
LIN {X 0,Y 585.849,Z 733.66,A -85,B 0,C 180,E1 1828.513,E2 1828.513} C_VEL
LIN {X 0,Y 585.876,Z 733.66,A -85,B 0,C 180,E1 1834.651,E2 1834.651} C_VEL
LIN {X 0,Y 585.77,Z 733.66,A -85,B 0,C 180,E1 1840.257,E2 1840.257} C_VEL
LIN {X 0,Y 585.941,Z 733.66,A -85,B 0,C 180,E1 1846.348,E2 1846.348} C_VEL
LIN {X 0,Y 585.836,Z 733.66,A -85,B 0,C 180,E1 1851.664,E2 1851.664} C_VEL
LIN {X 0,Y 585.732,Z 733.66,A -85,B 0,C 180,E1 1857.123,E2 1857.123} C_VEL
LIN {X 0,Y 585.833,Z 733.66,A -85,B 0,C 180,E1 1862.856,E2 1862.856} C_VEL
LIN {X 0,Y 586.059,Z 733.66,A -85,B 0,C 180,E1 1863.813,E2 1863.813} C_VEL
LIN {X 0,Y 589.17,Z 745.179,A -85,B 0,C 180,E1 1864.128,E2 1864.128} C_VEL
LIN {X 0,Y 588.975,Z 783.299,A -85,B 0,C 180,E1 1864.93,E2 1864.93} C_VEL
LIN {X 0,Y 588.509,Z 819.191,A -85,B 0,C 180,E1 1866.282,E2 1866.282} C_VEL
LIN {X 0,Y 587.93,Z 852.774,A -85,B 0,C 180,E1 1868.153,E2 1868.153} C_VEL
LIN {X 0,Y 587.449,Z 884.745,A -85,B 0,C 180,E1 1870.62,E2 1870.62} C_VEL
LIN {X 0,Y 586.956,Z 912.508,A -85,B 0,C 180,E1 1873.516,E2 1873.516} C_VEL
LIN {X 0,Y 586.682,Z 935.599,A -85,B 0,C 180,E1 1876.759,E2 1876.759} C_VEL
LIN {X 0,Y 586.519,Z 953.659,A -85,B 0,C 180,E1 1880.34,E2 1880.34} C_VEL
LIN {X 0,Y 586.444,Z 964.113,A -85,B 0,C 180,E1 1883.388,E2 1883.388} C_VEL
LIN {X 0,Y 586.396,Z 971.219,A -85,B 0,C 180,E1 1887.04,E2 1887.04} C_VEL
LIN {X 0,Y 586.353,Z 972.996,A -85,B 0,C 180,E1 1890,E2 1890} C_VEL
LIN {X 0,Y 586.456,Z 970.093,A -85,B 0,C 180,E1 1893.701,E2 1893.701} C_VEL
LIN {X 0,Y 586.449,Z 961.467,A -85,B 0,C 180,E1 1897.417,E2 1897.417} C_VEL
LIN {X 0,Y 586.545,Z 948.193,A -85,B 0,C 180,E1 1900.803,E2 1900.803} C_VEL
LIN {X 0,Y 586.766,Z 928.911,A -85,B 0,C 180,E1 1904.2,E2 1904.2} C_VEL
LIN {X 0,Y 587.094,Z 903.723,A -85,B 0,C 180,E1 1907.404,E2 1907.404} C_VEL
LIN {X 0,Y 587.622,Z 874.992,A -85,B 0,C 180,E1 1910.127,E2 1910.127} C_VEL
LIN {X 0,Y 588.135,Z 842.725,A -85,B 0,C 180,E1 1912.384,E2 1912.384} C_VEL
LIN {X 0,Y 588.644,Z 809.264,A -85,B 0,C 180,E1 1914.065,E2 1914.065} C_VEL
LIN {X 0,Y 589.12,Z 772.897,A -85,B 0,C 180,E1 1915.257,E2 1915.257} C_VEL
LIN {X 0,Y 588.5,Z 740.608,A -85,B 0,C 180,E1 1915.874,E2 1915.874} C_VEL
LIN {X 0,Y 586.291,Z 733.66,A -85,B 0,C 180,E1 1916.114,E2 1916.114} C_VEL
LIN {X 0,Y 585.946,Z 733.66,A -85,B 0,C 180,E1 1922.864,E2 1922.864} C_VEL
LIN {X 0,Y 585.795,Z 733.66,A -85,B 0,C 180,E1 1929.157,E2 1929.157} C_VEL
LIN {X 0,Y 585.839,Z 733.66,A -85,B 0,C 180,E1 1934.252,E2 1934.252} C_VEL
LIN {X 0,Y 585.826,Z 733.66,A -85,B 0,C 180,E1 1939.748,E2 1939.748} C_VEL
LIN {X 0,Y 585.811,Z 733.66,A -85,B 0,C 180,E1 1945.345,E2 1945.345} C_VEL
LIN {X 0,Y 585.86,Z 733.66,A -85,B 0,C 180,E1 1950.589,E2 1950.589} C_VEL
LIN {X 0,Y 585.991,Z 733.66,A -85,B 0,C 180,E1 1955.579,E2 1955.579} C_VEL
LIN {X 0,Y 586.136,Z 733.66,A -85,B 0,C 180,E1 1960.376,E2 1960.376} C_VEL
LIN {X 0,Y 585.822,Z 733.66,A -85,B 0,C 180,E1 1965.019,E2 1965.019} C_VEL
LIN {X 0,Y 586.112,Z 733.66,A -85,B 0,C 180,E1 1969.579,E2 1969.579} C_VEL
LIN {X 0,Y 586.303,Z 733.66,A -85,B 0,C 180,E1 1974.068,E2 1974.068} C_VEL
LIN {X 0,Y 586.104,Z 733.66,A -85,B 0,C 180,E1 1979.997,E2 1979.997} C_VEL
LIN {X 0,Y 586.144,Z 733.66,A -85,B 0,C 180,E1 1984.427,E2 1984.427} C_VEL
LIN {X 0,Y 583.681,Z 733.66,A -85,B 0,C 180,E1 1985.685,E2 1985.685} C_VEL
LIN {X 0,Y 578.288,Z 733.66,A -85,B 0,C 180,E1 1987.565,E2 1987.565} C_VEL
LIN {X 0,Y 578.18,Z 733.66,A -85,B 0,C 180,E1 1987.783,E2 1987.783} C_VEL
LIN {X 0,Y 578.228,Z 733.66,A -85,B 0,C 180,E1 1993.627,E2 1993.627} C_VEL
LIN {X 0,Y 578.115,Z 733.66,A -85,B 0,C 180,E1 1999.464,E2 1999.464} C_VEL
LIN {X 0,Y 577.971,Z 733.66,A -85,B 0,C 180,E1 2004.776,E2 2004.776} C_VEL
LIN {X 0,Y 577.838,Z 733.66,A -85,B 0,C 180,E1 2010.152,E2 2010.152} C_VEL
LIN {X 0,Y 577.852,Z 733.66,A -85,B 0,C 180,E1 2015.195,E2 2015.195} C_VEL
LIN {X 0,Y 577.833,Z 733.66,A -85,B 0,C 180,E1 2020.918,E2 2020.918} C_VEL
LIN {X 0,Y 577.987,Z 733.66,A -85,B 0,C 180,E1 2027.171,E2 2027.171} C_VEL
LIN {X 0,Y 577.969,Z 733.66,A -85,B 0,C 180,E1 2032.949,E2 2032.949} C_VEL
LIN {X 0,Y 577.919,Z 733.66,A -85,B 0,C 180,E1 2038.4,E2 2038.4} C_VEL
LIN {X 0,Y 578.113,Z 734.188,A -85,B 0,C 180,E1 2042.81,E2 2042.81} C_VEL
LIN {X 0,Y 582.004,Z 745.749,A -85,B 0,C 180,E1 2043.163,E2 2043.163} C_VEL
LIN {X 0,Y 581.961,Z 819.424,A -85,B 0,C 180,E1 2044.277,E2 2044.277} C_VEL
LIN {X 0,Y 581.447,Z 856.314,A -85,B 0,C 180,E1 2045.446,E2 2045.446} C_VEL
LIN {X 0,Y 580.723,Z 891.503,A -85,B 0,C 180,E1 2047.193,E2 2047.193} C_VEL
LIN {X 0,Y 580.026,Z 923.954,A -85,B 0,C 180,E1 2049.466,E2 2049.466} C_VEL
LIN {X 0,Y 579.39,Z 953.024,A -85,B 0,C 180,E1 2052.234,E2 2052.234} C_VEL
LIN {X 0,Y 578.937,Z 977.594,A -85,B 0,C 180,E1 2055.363,E2 2055.363} C_VEL
LIN {X 0,Y 578.63,Z 996.454,A -85,B 0,C 180,E1 2058.632,E2 2058.632} C_VEL
LIN {X 0,Y 578.52,Z 1010.447,A -85,B 0,C 180,E1 2062.102,E2 2062.102} C_VEL
LIN {X 0,Y 578.413,Z 1018.973,A -85,B 0,C 180,E1 2065.496,E2 2065.496} C_VEL
LIN {X 0,Y 578.418,Z 1022.516,A -85,B 0,C 180,E1 2068.5,E2 2068.5} C_VEL
LIN {X 0,Y 578.498,Z 1022.516,A -85,B 0,C 180,E1 2071.5,E2 2071.5} C_VEL
LIN {X 0,Y 578.515,Z 1017.49,A -85,B 0,C 180,E1 2075.24,E2 2075.24} C_VEL
LIN {X 0,Y 578.541,Z 1007.847,A -85,B 0,C 180,E1 2078.655,E2 2078.655} C_VEL
LIN {X 0,Y 578.709,Z 991.837,A -85,B 0,C 180,E1 2082.273,E2 2082.273} C_VEL
LIN {X 0,Y 579.048,Z 969.749,A -85,B 0,C 180,E1 2085.741,E2 2085.741} C_VEL
LIN {X 0,Y 579.564,Z 944.495,A -85,B 0,C 180,E1 2088.664,E2 2088.664} C_VEL
LIN {X 0,Y 580.234,Z 913.89,A -85,B 0,C 180,E1 2091.317,E2 2091.317} C_VEL
LIN {X 0,Y 580.989,Z 880.745,A -85,B 0,C 180,E1 2093.411,E2 2093.411} C_VEL
LIN {X 0,Y 581.64,Z 845.271,A -85,B 0,C 180,E1 2094.969,E2 2094.969} C_VEL
LIN {X 0,Y 582.085,Z 809.454,A -85,B 0,C 180,E1 2095.931,E2 2095.931} C_VEL
LIN {X 0,Y 581.484,Z 743.551,A -85,B 0,C 180,E1 2096.892,E2 2096.892} C_VEL
LIN {X 0,Y 578.104,Z 733.66,A -85,B 0,C 180,E1 2097.224,E2 2097.224} C_VEL
LIN {X 0,Y 577.844,Z 733.66,A -85,B 0,C 180,E1 2103.031,E2 2103.031} C_VEL
LIN {X 0,Y 577.9,Z 733.66,A -85,B 0,C 180,E1 2108.961,E2 2108.961} C_VEL
LIN {X 0,Y 577.941,Z 733.66,A -85,B 0,C 180,E1 2115.019,E2 2115.019} C_VEL
LIN {X 0,Y 577.879,Z 733.66,A -85,B 0,C 180,E1 2121.044,E2 2121.044} C_VEL
LIN {X 0,Y 578.086,Z 733.66,A -85,B 0,C 180,E1 2126.943,E2 2126.943} C_VEL
LIN {X 0,Y 577.869,Z 733.66,A -85,B 0,C 180,E1 2132.979,E2 2132.979} C_VEL
LIN {X 0,Y 577.916,Z 733.66,A -85,B 0,C 180,E1 2138.487,E2 2138.487} C_VEL
LIN {X 0,Y 578.164,Z 733.66,A -85,B 0,C 180,E1 2141.431,E2 2141.431} C_VEL
LIN {X 0,Y 579.767,Z 760.263,A -85,B 0,C 180,E1 2142.013,E2 2142.013} C_VEL
LIN {X 0,Y 579.453,Z 788.361,A -85,B 0,C 180,E1 2143.142,E2 2143.142} C_VEL
LIN {X 0,Y 579.178,Z 813.372,A -85,B 0,C 180,E1 2144.753,E2 2144.753} C_VEL
LIN {X 0,Y 578.892,Z 834.529,A -85,B 0,C 180,E1 2146.774,E2 2146.774} C_VEL
LIN {X 0,Y 578.69,Z 852.4,A -85,B 0,C 180,E1 2149.279,E2 2149.279} C_VEL
LIN {X 0,Y 578.596,Z 863.775,A -85,B 0,C 180,E1 2151.729,E2 2151.729} C_VEL
LIN {X 0,Y 578.58,Z 871.348,A -85,B 0,C 180,E1 2154.748,E2 2154.748} C_VEL
LIN {X 0,Y 578.485,Z 872.958,A -85,B 0,C 180,E1 2157.003,E2 2157.003} C_VEL
LIN {X 0,Y 578.502,Z 869.907,A -85,B 0,C 180,E1 2160.003,E2 2160.003} C_VEL
LIN {X 0,Y 578.571,Z 862.054,A -85,B 0,C 180,E1 2162.628,E2 2162.628} C_VEL
LIN {X 0,Y 578.725,Z 848.606,A -85,B 0,C 180,E1 2165.257,E2 2165.257} C_VEL
LIN {X 0,Y 578.93,Z 831.146,A -85,B 0,C 180,E1 2167.517,E2 2167.517} C_VEL
LIN {X 0,Y 579.214,Z 807.505,A -85,B 0,C 180,E1 2169.596,E2 2169.596} C_VEL
LIN {X 0,Y 579.579,Z 780.757,A -85,B 0,C 180,E1 2171.14,E2 2171.14} C_VEL
LIN {X 0,Y 579.854,Z 751.998,A -85,B 0,C 180,E1 2172.108,E2 2172.108} C_VEL
LIN {X 0,Y 578.36,Z 733.66,A -85,B 0,C 180,E1 2172.476,E2 2172.476} C_VEL
LIN {X 0,Y 578.148,Z 733.66,A -85,B 0,C 180,E1 2178.319,E2 2178.319} C_VEL
LIN {X 0,Y 578.004,Z 733.66,A -85,B 0,C 180,E1 2183.533,E2 2183.533} C_VEL
LIN {X 0,Y 577.976,Z 733.66,A -85,B 0,C 180,E1 2188.136,E2 2188.136} C_VEL
LIN {X 0,Y 578.037,Z 733.66,A -85,B 0,C 180,E1 2193.374,E2 2193.374} C_VEL
LIN {X 0,Y 577.88,Z 733.66,A -85,B 0,C 180,E1 2198.965,E2 2198.965} C_VEL
LIN {X 0,Y 577.97,Z 733.66,A -85,B 0,C 180,E1 2205.018,E2 2205.018} C_VEL
LIN {X 0,Y 577.92,Z 733.66,A -85,B 0,C 180,E1 2211.04,E2 2211.04} C_VEL
LIN {X 0,Y 577.843,Z 733.66,A -85,B 0,C 180,E1 2216.981,E2 2216.981} C_VEL
LIN {X 0,Y 577.974,Z 733.66,A -85,B 0,C 180,E1 2222.96,E2 2222.96} C_VEL
LIN {X 0,Y 578.068,Z 733.66,A -85,B 0,C 180,E1 2223.436,E2 2223.436} C_VEL
LIN {X 0,Y 581.946,Z 744.445,A -85,B 0,C 180,E1 2223.773,E2 2223.773} C_VEL
LIN {X 0,Y 581.825,Z 783.289,A -85,B 0,C 180,E1 2224.6,E2 2224.6} C_VEL
LIN {X 0,Y 581.201,Z 819.703,A -85,B 0,C 180,E1 2225.99,E2 2225.99} C_VEL
LIN {X 0,Y 580.446,Z 854.121,A -85,B 0,C 180,E1 2227.948,E2 2227.948} C_VEL
LIN {X 0,Y 579.824,Z 885.786,A -85,B 0,C 180,E1 2230.454,E2 2230.454} C_VEL
LIN {X 0,Y 579.196,Z 912.506,A -85,B 0,C 180,E1 2233.289,E2 2233.289} C_VEL
LIN {X 0,Y 578.86,Z 935.595,A -85,B 0,C 180,E1 2236.577,E2 2236.577} C_VEL
LIN {X 0,Y 578.656,Z 953.658,A -85,B 0,C 180,E1 2240.208,E2 2240.208} C_VEL
LIN {X 0,Y 578.553,Z 963.959,A -85,B 0,C 180,E1 2243.237,E2 2243.237} C_VEL
LIN {X 0,Y 578.495,Z 971.218,A -85,B 0,C 180,E1 2247,E2 2247} C_VEL
LIN {X 0,Y 578.453,Z 972.997,A -85,B 0,C 180,E1 2250,E2 2250} C_VEL
LIN {X 0,Y 578.569,Z 970.094,A -85,B 0,C 180,E1 2253.751,E2 2253.751} C_VEL
LIN {X 0,Y 578.571,Z 961.47,A -85,B 0,C 180,E1 2257.519,E2 2257.519} C_VEL
LIN {X 0,Y 578.681,Z 948.198,A -85,B 0,C 180,E1 2260.952,E2 2260.952} C_VEL
LIN {X 0,Y 578.961,Z 928.33,A -85,B 0,C 180,E1 2264.481,E2 2264.481} C_VEL
LIN {X 0,Y 579.408,Z 903.731,A -85,B 0,C 180,E1 2267.642,E2 2267.642} C_VEL
LIN {X 0,Y 580.034,Z 874.61,A -85,B 0,C 180,E1 2270.434,E2 2270.434} C_VEL
LIN {X 0,Y 580.709,Z 842.732,A -85,B 0,C 180,E1 2272.687,E2 2272.687} C_VEL
LIN {X 0,Y 581.418,Z 808.683,A -85,B 0,C 180,E1 2274.409,E2 2274.409} C_VEL
LIN {X 0,Y 581.968,Z 771.717,A -85,B 0,C 180,E1 2275.621,E2 2275.621} C_VEL
LIN {X 0,Y 581.405,Z 742.642,A -85,B 0,C 180,E1 2276.187,E2 2276.187} C_VEL
LIN {X 0,Y 578.369,Z 733.66,A -85,B 0,C 180,E1 2276.508,E2 2276.508} C_VEL
LIN {X 0,Y 578.033,Z 733.66,A -85,B 0,C 180,E1 2283.372,E2 2283.372} C_VEL
LIN {X 0,Y 577.879,Z 733.66,A -85,B 0,C 180,E1 2288.963,E2 2288.963} C_VEL
LIN {X 0,Y 577.929,Z 733.66,A -85,B 0,C 180,E1 2295.021,E2 2295.021} C_VEL
LIN {X 0,Y 577.882,Z 733.66,A -85,B 0,C 180,E1 2301.035,E2 2301.035} C_VEL
LIN {X 0,Y 577.832,Z 733.66,A -85,B 0,C 180,E1 2306.982,E2 2306.982} C_VEL
LIN {X 0,Y 577.936,Z 733.66,A -85,B 0,C 180,E1 2312.967,E2 2312.967} C_VEL
LIN {X 0,Y 578.084,Z 733.66,A -85,B 0,C 180,E1 2318.487,E2 2318.487} C_VEL
LIN {X 0,Y 578.225,Z 733.66,A -85,B 0,C 180,E1 2323.257,E2 2323.257} C_VEL
LIN {X 0,Y 578.185,Z 733.66,A -85,B 0,C 180,E1 2329.435,E2 2329.435} C_VEL
LIN {X 0,Y 578.396,Z 733.66,A -85,B 0,C 180,E1 2334.125,E2 2334.125} C_VEL
LIN {X 0,Y 578.203,Z 733.66,A -85,B 0,C 180,E1 2339.997,E2 2339.997} C_VEL
LIN {X 0,Y 578.229,Z 733.66,A -85,B 0,C 180,E1 2344.502,E2 2344.502} C_VEL
LIN {X 0,Y 578.18,Z 733.66,A -85,B 0,C 180,E1 2347.783,E2 2347.783} C_VEL
LIN {X 0,Y 574.145,Z 733.66,A -85,B 0,C 180,E1 2349.472,E2 2349.472} C_VEL
LIN {X 0,Y 570.162,Z 733.66,A -85,B 0,C 180,E1 2351.184,E2 2351.184} C_VEL
LIN {X 0,Y 570.111,Z 733.66,A -85,B 0,C 180,E1 2355.397,E2 2355.397} C_VEL
LIN {X 0,Y 570.132,Z 733.66,A -85,B 0,C 180,E1 2360.192,E2 2360.192} C_VEL
LIN {X 0,Y 570.019,Z 733.66,A -85,B 0,C 180,E1 2365.429,E2 2365.429} C_VEL
LIN {X 0,Y 569.954,Z 733.66,A -85,B 0,C 180,E1 2370.308,E2 2370.308} C_VEL
LIN {X 0,Y 569.91,Z 733.66,A -85,B 0,C 180,E1 2375.76,E2 2375.76} C_VEL
LIN {X 0,Y 569.872,Z 733.66,A -85,B 0,C 180,E1 2381.615,E2 2381.615} C_VEL
LIN {X 0,Y 569.986,Z 733.66,A -85,B 0,C 180,E1 2386.318,E2 2386.318} C_VEL
LIN {X 0,Y 570.049,Z 733.66,A -85,B 0,C 180,E1 2392.345,E2 2392.345} C_VEL
LIN {X 0,Y 570.001,Z 733.66,A -85,B 0,C 180,E1 2398.202,E2 2398.202} C_VEL
LIN {X 0,Y 570.147,Z 733.822,A -85,B 0,C 180,E1 2402.393,E2 2402.393} C_VEL
LIN {X 0,Y 575.077,Z 749.158,A -85,B 0,C 180,E1 2402.861,E2 2402.861} C_VEL
LIN {X 0,Y 574.835,Z 820.13,A -85,B 0,C 180,E1 2403.952,E2 2403.952} C_VEL
LIN {X 0,Y 574.179,Z 857.133,A -85,B 0,C 180,E1 2405.149,E2 2405.149} C_VEL
LIN {X 0,Y 573.315,Z 892.617,A -85,B 0,C 180,E1 2406.949,E2 2406.949} C_VEL
LIN {X 0,Y 572.441,Z 925.131,A -85,B 0,C 180,E1 2409.282,E2 2409.282} C_VEL
LIN {X 0,Y 571.712,Z 953.54,A -85,B 0,C 180,E1 2412.046,E2 2412.046} C_VEL
LIN {X 0,Y 571.141,Z 978.59,A -85,B 0,C 180,E1 2415.308,E2 2415.308} C_VEL
LIN {X 0,Y 570.773,Z 997.837,A -85,B 0,C 180,E1 2418.767,E2 2418.767} C_VEL
LIN {X 0,Y 570.606,Z 1011.609,A -85,B 0,C 180,E1 2422.376,E2 2422.376} C_VEL
LIN {X 0,Y 570.545,Z 1020.18,A -85,B 0,C 180,E1 2426.196,E2 2426.196} C_VEL
LIN {X 0,Y 570.496,Z 1023,A -85,B 0,C 180,E1 2430,E2 2430} C_VEL
LIN {X 0,Y 570.624,Z 1020.181,A -85,B 0,C 180,E1 2433.803,E2 2433.803} C_VEL
LIN {X 0,Y 570.654,Z 1011.608,A -85,B 0,C 180,E1 2437.623,E2 2437.623} C_VEL
LIN {X 0,Y 570.861,Z 997.804,A -85,B 0,C 180,E1 2441.239,E2 2441.239} C_VEL
LIN {X 0,Y 571.179,Z 977.447,A -85,B 0,C 180,E1 2444.862,E2 2444.862} C_VEL
LIN {X 0,Y 571.738,Z 952.613,A -85,B 0,C 180,E1 2448.058,E2 2448.058} C_VEL
LIN {X 0,Y 572.543,Z 922.713,A -85,B 0,C 180,E1 2450.916,E2 2450.916} C_VEL
LIN {X 0,Y 573.394,Z 890.55,A -85,B 0,C 180,E1 2453.174,E2 2453.174} C_VEL
LIN {X 0,Y 574.178,Z 854.652,A -85,B 0,C 180,E1 2454.955,E2 2454.955} C_VEL
LIN {X 0,Y 574.859,Z 816.531,A -85,B 0,C 180,E1 2456.133,E2 2456.133} C_VEL
LIN {X 0,Y 574.299,Z 745.078,A -85,B 0,C 180,E1 2457.235,E2 2457.235} C_VEL
LIN {X 0,Y 570.146,Z 733.66,A -85,B 0,C 180,E1 2457.638,E2 2457.638} C_VEL
LIN {X 0,Y 569.965,Z 733.66,A -85,B 0,C 180,E1 2462.093,E2 2462.093} C_VEL
LIN {X 0,Y 570.019,Z 733.66,A -85,B 0,C 180,E1 2467.656,E2 2467.656} C_VEL
LIN {X 0,Y 569.984,Z 733.66,A -85,B 0,C 180,E1 2473.682,E2 2473.682} C_VEL
LIN {X 0,Y 569.869,Z 733.66,A -85,B 0,C 180,E1 2478.384,E2 2478.384} C_VEL
LIN {X 0,Y 569.92,Z 733.66,A -85,B 0,C 180,E1 2484.241,E2 2484.241} C_VEL
LIN {X 0,Y 570.072,Z 733.66,A -85,B 0,C 180,E1 2489.699,E2 2489.699} C_VEL
LIN {X 0,Y 569.959,Z 733.66,A -85,B 0,C 180,E1 2494.852,E2 2494.852} C_VEL
LIN {X 0,Y 570.25,Z 733.66,A -85,B 0,C 180,E1 2501.208,E2 2501.208} C_VEL
LIN {X 0,Y 572.135,Z 758.447,A -85,B 0,C 180,E1 2501.757,E2 2501.757} C_VEL
LIN {X 0,Y 571.802,Z 785.696,A -85,B 0,C 180,E1 2502.813,E2 2502.813} C_VEL
LIN {X 0,Y 571.414,Z 811.526,A -85,B 0,C 180,E1 2504.442,E2 2504.442} C_VEL
LIN {X 0,Y 571.104,Z 832.5,A -85,B 0,C 180,E1 2506.395,E2 2506.395} C_VEL
LIN {X 0,Y 570.838,Z 850.954,A -85,B 0,C 180,E1 2508.928,E2 2508.928} C_VEL
LIN {X 0,Y 570.715,Z 863.629,A -85,B 0,C 180,E1 2511.614,E2 2511.614} C_VEL
LIN {X 0,Y 570.692,Z 870.006,A -85,B 0,C 180,E1 2513.912,E2 2513.912} C_VEL
LIN {X 0,Y 570.582,Z 872.947,A -85,B 0,C 180,E1 2516.961,E2 2516.961} C_VEL
LIN {X 0,Y 570.632,Z 869.996,A -85,B 0,C 180,E1 2520.003,E2 2520.003} C_VEL
LIN {X 0,Y 570.689,Z 862.219,A -85,B 0,C 180,E1 2522.664,E2 2522.664} C_VEL
LIN {X 0,Y 570.901,Z 847.879,A -85,B 0,C 180,E1 2525.487,E2 2525.487} C_VEL
LIN {X 0,Y 571.112,Z 829.732,A -85,B 0,C 180,E1 2527.812,E2 2527.812} C_VEL
LIN {X 0,Y 571.486,Z 805.467,A -85,B 0,C 180,E1 2529.919,E2 2529.919} C_VEL
LIN {X 0,Y 571.905,Z 779.411,A -85,B 0,C 180,E1 2531.392,E2 2531.392} C_VEL
LIN {X 0,Y 572.237,Z 751.471,A -85,B 0,C 180,E1 2532.327,E2 2532.327} C_VEL
LIN {X 0,Y 570.417,Z 733.66,A -85,B 0,C 180,E1 2532.732,E2 2532.732} C_VEL
LIN {X 0,Y 570.221,Z 733.66,A -85,B 0,C 180,E1 2538.583,E2 2538.583} C_VEL
LIN {X 0,Y 570.128,Z 733.66,A -85,B 0,C 180,E1 2543.478,E2 2543.478} C_VEL
LIN {X 0,Y 569.992,Z 733.66,A -85,B 0,C 180,E1 2548.766,E2 2548.766} C_VEL
LIN {X 0,Y 569.953,Z 733.66,A -85,B 0,C 180,E1 2554.562,E2 2554.562} C_VEL
LIN {X 0,Y 569.921,Z 733.66,A -85,B 0,C 180,E1 2559.615,E2 2559.615} C_VEL
LIN {X 0,Y 569.989,Z 733.66,A -85,B 0,C 180,E1 2565.827,E2 2565.827} C_VEL
LIN {X 0,Y 570.007,Z 733.66,A -85,B 0,C 180,E1 2570.394,E2 2570.394} C_VEL
LIN {X 0,Y 569.884,Z 733.66,A -85,B 0,C 180,E1 2576.087,E2 2576.087} C_VEL
LIN {X 0,Y 569.927,Z 733.66,A -85,B 0,C 180,E1 2581.433,E2 2581.433} C_VEL
LIN {X 0,Y 570.081,Z 733.69,A -85,B 0,C 180,E1 2583.037,E2 2583.037} C_VEL
LIN {X 0,Y 574.972,Z 748.655,A -85,B 0,C 180,E1 2583.492,E2 2583.492} C_VEL
LIN {X 0,Y 574.564,Z 787.055,A -85,B 0,C 180,E1 2584.376,E2 2584.376} C_VEL
LIN {X 0,Y 573.817,Z 822.715,A -85,B 0,C 180,E1 2585.81,E2 2585.81} C_VEL
LIN {X 0,Y 572.957,Z 856.8,A -85,B 0,C 180,E1 2587.829,E2 2587.829} C_VEL
LIN {X 0,Y 572.135,Z 888.282,A -85,B 0,C 180,E1 2590.421,E2 2590.421} C_VEL
LIN {X 0,Y 571.416,Z 915.666,A -85,B 0,C 180,E1 2593.451,E2 2593.451} C_VEL
LIN {X 0,Y 571.005,Z 937.789,A -85,B 0,C 180,E1 2596.78,E2 2596.78} C_VEL
LIN {X 0,Y 570.766,Z 953.657,A -85,B 0,C 180,E1 2600.071,E2 2600.071} C_VEL
LIN {X 0,Y 570.649,Z 963.958,A -85,B 0,C 180,E1 2603.143,E2 2603.143} C_VEL
LIN {X 0,Y 570.594,Z 971.218,A -85,B 0,C 180,E1 2606.958,E2 2606.958} C_VEL
LIN {X 0,Y 570.553,Z 972.997,A -85,B 0,C 180,E1 2610,E2 2610} C_VEL
LIN {X 0,Y 570.659,Z 970.095,A -85,B 0,C 180,E1 2613.804,E2 2613.804} C_VEL
LIN {X 0,Y 570.674,Z 961.473,A -85,B 0,C 180,E1 2617.623,E2 2617.623} C_VEL
LIN {X 0,Y 570.815,Z 947.603,A -85,B 0,C 180,E1 2621.237,E2 2621.237} C_VEL
LIN {X 0,Y 571.177,Z 927.327,A -85,B 0,C 180,E1 2624.834,E2 2624.834} C_VEL
LIN {X 0,Y 571.723,Z 903.179,A -85,B 0,C 180,E1 2627.951,E2 2627.951} C_VEL
LIN {X 0,Y 572.512,Z 873.365,A -85,B 0,C 180,E1 2630.817,E2 2630.817} C_VEL
LIN {X 0,Y 573.361,Z 840.796,A -85,B 0,C 180,E1 2633.113,E2 2633.113} C_VEL
LIN {X 0,Y 574.29,Z 806.167,A -85,B 0,C 180,E1 2634.841,E2 2634.841} C_VEL
LIN {X 0,Y 574.878,Z 770.82,A -85,B 0,C 180,E1 2635.986,E2 2635.986} C_VEL
LIN {X 0,Y 574.393,Z 744.892,A -85,B 0,C 180,E1 2636.501,E2 2636.501} C_VEL
LIN {X 0,Y 570.398,Z 733.66,A -85,B 0,C 180,E1 2636.9,E2 2636.9} C_VEL
LIN {X 0,Y 570.02,Z 733.66,A -85,B 0,C 180,E1 2642.09,E2 2642.09} C_VEL
LIN {X 0,Y 569.917,Z 733.66,A -85,B 0,C 180,E1 2647.665,E2 2647.665} C_VEL
LIN {X 0,Y 569.892,Z 733.66,A -85,B 0,C 180,E1 2653.691,E2 2653.691} C_VEL
LIN {X 0,Y 569.973,Z 733.66,A -85,B 0,C 180,E1 2658.384,E2 2658.384} C_VEL
LIN {X 0,Y 569.979,Z 733.66,A -85,B 0,C 180,E1 2664.237,E2 2664.237} C_VEL
LIN {X 0,Y 569.997,Z 733.66,A -85,B 0,C 180,E1 2669.686,E2 2669.686} C_VEL
LIN {X 0,Y 570.147,Z 733.66,A -85,B 0,C 180,E1 2674.853,E2 2674.853} C_VEL
LIN {X 0,Y 570.242,Z 733.66,A -85,B 0,C 180,E1 2679.805,E2 2679.805} C_VEL
LIN {X 0,Y 570.057,Z 733.66,A -85,B 0,C 180,E1 2684.595,E2 2684.595} C_VEL
LIN {X 0,Y 570.167,Z 733.66,A -85,B 0,C 180,E1 2690.829,E2 2690.829} C_VEL
LIN {X 0,Y 570.247,Z 733.66,A -85,B 0,C 180,E1 2695.428,E2 2695.428} C_VEL
LIN {X 0,Y 570.315,Z 733.66,A -85,B 0,C 180,E1 2699.997,E2 2699.997} C_VEL
LIN {X 0,Y 570.327,Z 733.66,A -85,B 0,C 180,E1 2704.564,E2 2704.564} C_VEL
LIN {X 0,Y 570.295,Z 733.66,A -85,B 0,C 180,E1 2709.162,E2 2709.162} C_VEL
LIN {X 0,Y 570.162,Z 733.66,A -85,B 0,C 180,E1 2711.184,E2 2711.184} C_VEL
LIN {X 0,Y 568.934,Z 733.66,A -85,B 0,C 180,E1 2712.052,E2 2712.052} C_VEL
LIN {X 0,Y 562.357,Z 733.66,A -85,B 0,C 180,E1 2714.413,E2 2714.413} C_VEL
LIN {X 0,Y 562.241,Z 733.66,A -85,B 0,C 180,E1 2714.637,E2 2714.637} C_VEL
LIN {X 0,Y 562.249,Z 733.66,A -85,B 0,C 180,E1 2719.52,E2 2719.52} C_VEL
LIN {X 0,Y 562.123,Z 733.66,A -85,B 0,C 180,E1 2725.523,E2 2725.523} C_VEL
LIN {X 0,Y 562.038,Z 733.66,A -85,B 0,C 180,E1 2730.781,E2 2730.781} C_VEL
LIN {X 0,Y 561.994,Z 733.66,A -85,B 0,C 180,E1 2736.343,E2 2736.343} C_VEL
LIN {X 0,Y 561.952,Z 733.66,A -85,B 0,C 180,E1 2742.337,E2 2742.337} C_VEL
LIN {X 0,Y 562.061,Z 733.66,A -85,B 0,C 180,E1 2747.665,E2 2747.665} C_VEL
LIN {X 0,Y 562.104,Z 733.66,A -85,B 0,C 180,E1 2753.899,E2 2753.899} C_VEL
LIN {X 0,Y 562.135,Z 733.66,A -85,B 0,C 180,E1 2759.519,E2 2759.519} C_VEL
LIN {X 0,Y 562.239,Z 733.66,A -85,B 0,C 180,E1 2761.955,E2 2761.955} C_VEL
LIN {X 0,Y 568.072,Z 751.465,A -85,B 0,C 180,E1 2762.53,E2 2762.53} C_VEL
LIN {X 0,Y 567.721,Z 820.48,A -85,B 0,C 180,E1 2763.609,E2 2763.609} C_VEL
LIN {X 0,Y 566.982,Z 856.97,A -85,B 0,C 180,E1 2764.804,E2 2764.804} C_VEL
LIN {X 0,Y 565.966,Z 891.845,A -85,B 0,C 180,E1 2766.584,E2 2766.584} C_VEL
LIN {X 0,Y 564.907,Z 925.127,A -85,B 0,C 180,E1 2768.993,E2 2768.993} C_VEL
LIN {X 0,Y 564.014,Z 953.974,A -85,B 0,C 180,E1 2771.843,E2 2771.843} C_VEL
LIN {X 0,Y 563.366,Z 977.678,A -85,B 0,C 180,E1 2774.961,E2 2774.961} C_VEL
LIN {X 0,Y 562.943,Z 996.695,A -85,B 0,C 180,E1 2778.362,E2 2778.362} C_VEL
LIN {X 0,Y 562.76,Z 1010.439,A -85,B 0,C 180,E1 2781.88,E2 2781.88} C_VEL
LIN {X 0,Y 562.65,Z 1018.968,A -85,B 0,C 180,E1 2785.369,E2 2785.369} C_VEL
LIN {X 0,Y 562.622,Z 1022.52,A -85,B 0,C 180,E1 2788.458,E2 2788.458} C_VEL
LIN {X 0,Y 562.695,Z 1022.52,A -85,B 0,C 180,E1 2791.542,E2 2791.542} C_VEL
LIN {X 0,Y 562.694,Z 1017.366,A -85,B 0,C 180,E1 2795.452,E2 2795.452} C_VEL
LIN {X 0,Y 562.782,Z 1006.476,A -85,B 0,C 180,E1 2799.289,E2 2799.289} C_VEL
LIN {X 0,Y 563.048,Z 990.786,A -85,B 0,C 180,E1 2802.818,E2 2802.818} C_VEL
LIN {X 0,Y 563.505,Z 969.759,A -85,B 0,C 180,E1 2806.186,E2 2806.186} C_VEL
LIN {X 0,Y 564.321,Z 943.261,A -85,B 0,C 180,E1 2809.316,E2 2809.316} C_VEL
LIN {X 0,Y 565.316,Z 913.759,A -85,B 0,C 180,E1 2811.918,E2 2811.918} C_VEL
LIN {X 0,Y 566.366,Z 880.839,A -85,B 0,C 180,E1 2814.048,E2 2814.048} C_VEL
LIN {X 0,Y 567.245,Z 846.25,A -85,B 0,C 180,E1 2815.612,E2 2815.612} C_VEL
LIN {X 0,Y 567.896,Z 810.193,A -85,B 0,C 180,E1 2816.614,E2 2816.614} C_VEL
LIN {X 0,Y 567.298,Z 747.281,A -85,B 0,C 180,E1 2817.569,E2 2817.569} C_VEL
LIN {X 0,Y 562.207,Z 733.66,A -85,B 0,C 180,E1 2818.09,E2 2818.09} C_VEL
LIN {X 0,Y 561.954,Z 733.66,A -85,B 0,C 180,E1 2823.37,E2 2823.37} C_VEL
LIN {X 0,Y 562.043,Z 733.66,A -85,B 0,C 180,E1 2828.636,E2 2828.636} C_VEL
LIN {X 0,Y 562.058,Z 733.66,A -85,B 0,C 180,E1 2834.459,E2 2834.459} C_VEL
LIN {X 0,Y 561.965,Z 733.66,A -85,B 0,C 180,E1 2839.719,E2 2839.719} C_VEL
LIN {X 0,Y 562.073,Z 733.66,A -85,B 0,C 180,E1 2845.556,E2 2845.556} C_VEL
LIN {X 0,Y 562.115,Z 733.66,A -85,B 0,C 180,E1 2851.004,E2 2851.004} C_VEL
LIN {X 0,Y 562.121,Z 733.66,A -85,B 0,C 180,E1 2856.319,E2 2856.319} C_VEL
LIN {X 0,Y 562.354,Z 733.66,A -85,B 0,C 180,E1 2860.985,E2 2860.985} C_VEL
LIN {X 0,Y 564.49,Z 755.029,A -85,B 0,C 180,E1 2861.459,E2 2861.459} C_VEL
LIN {X 0,Y 564.181,Z 783.494,A -85,B 0,C 180,E1 2862.503,E2 2862.503} C_VEL
LIN {X 0,Y 563.704,Z 809.611,A -85,B 0,C 180,E1 2864.124,E2 2864.124} C_VEL
LIN {X 0,Y 563.281,Z 832.109,A -85,B 0,C 180,E1 2866.203,E2 2866.203} C_VEL
LIN {X 0,Y 562.956,Z 850.681,A -85,B 0,C 180,E1 2868.771,E2 2868.771} C_VEL
LIN {X 0,Y 562.828,Z 863.482,A -85,B 0,C 180,E1 2871.495,E2 2871.495} C_VEL
LIN {X 0,Y 562.786,Z 871.075,A -85,B 0,C 180,E1 2874.519,E2 2874.519} C_VEL
LIN {X 0,Y 562.679,Z 872.937,A -85,B 0,C 180,E1 2876.919,E2 2876.919} C_VEL
LIN {X 0,Y 562.734,Z 870.085,A -85,B 0,C 180,E1 2880.003,E2 2880.003} C_VEL
LIN {X 0,Y 562.815,Z 862.385,A -85,B 0,C 180,E1 2882.702,E2 2882.702} C_VEL
LIN {X 0,Y 563.046,Z 847.868,A -85,B 0,C 180,E1 2885.609,E2 2885.609} C_VEL
LIN {X 0,Y 563.307,Z 830.134,A -85,B 0,C 180,E1 2887.921,E2 2887.921} C_VEL
LIN {X 0,Y 563.739,Z 806.045,A -85,B 0,C 180,E1 2890.057,E2 2890.057} C_VEL
LIN {X 0,Y 564.234,Z 780.373,A -85,B 0,C 180,E1 2891.549,E2 2891.549} C_VEL
LIN {X 0,Y 564.633,Z 751.485,A -85,B 0,C 180,E1 2892.538,E2 2892.538} C_VEL
LIN {X 0,Y 562.46,Z 733.66,A -85,B 0,C 180,E1 2892.933,E2 2892.933} C_VEL
LIN {X 0,Y 562.272,Z 733.66,A -85,B 0,C 180,E1 2898.855,E2 2898.855} C_VEL
LIN {X 0,Y 562.173,Z 733.66,A -85,B 0,C 180,E1 2903.83,E2 2903.83} C_VEL
LIN {X 0,Y 562.058,Z 733.66,A -85,B 0,C 180,E1 2909.008,E2 2909.008} C_VEL
LIN {X 0,Y 562.063,Z 733.66,A -85,B 0,C 180,E1 2914.453,E2 2914.453} C_VEL
LIN {X 0,Y 561.924,Z 733.66,A -85,B 0,C 180,E1 2920.293,E2 2920.293} C_VEL
LIN {X 0,Y 562.077,Z 733.66,A -85,B 0,C 180,E1 2925.543,E2 2925.543} C_VEL
LIN {X 0,Y 562.034,Z 733.66,A -85,B 0,C 180,E1 2931.713,E2 2931.713} C_VEL
LIN {X 0,Y 561.967,Z 733.66,A -85,B 0,C 180,E1 2937.395,E2 2937.395} C_VEL
LIN {X 0,Y 562.14,Z 733.66,A -85,B 0,C 180,E1 2942.615,E2 2942.615} C_VEL
LIN {X 0,Y 567.868,Z 750.191,A -85,B 0,C 180,E1 2943.16,E2 2943.16} C_VEL
LIN {X 0,Y 567.411,Z 787.044,A -85,B 0,C 180,E1 2944.029,E2 2944.029} C_VEL
LIN {X 0,Y 566.543,Z 823.304,A -85,B 0,C 180,E1 2945.51,E2 2945.51} C_VEL
LIN {X 0,Y 565.458,Z 858.339,A -85,B 0,C 180,E1 2947.635,E2 2947.635} C_VEL
LIN {X 0,Y 564.558,Z 888.419,A -85,B 0,C 180,E1 2950.161,E2 2950.161} C_VEL
LIN {X 0,Y 563.671,Z 915.661,A -85,B 0,C 180,E1 2953.217,E2 2953.217} C_VEL
LIN {X 0,Y 563.176,Z 937.788,A -85,B 0,C 180,E1 2956.592,E2 2956.592} C_VEL
LIN {X 0,Y 562.907,Z 953.655,A -85,B 0,C 180,E1 2959.931,E2 2959.931} C_VEL
LIN {X 0,Y 562.775,Z 963.957,A -85,B 0,C 180,E1 2963.046,E2 2963.046} C_VEL
LIN {X 0,Y 562.693,Z 971.217,A -85,B 0,C 180,E1 2966.915,E2 2966.915} C_VEL
LIN {X 0,Y 562.653,Z 972.997,A -85,B 0,C 180,E1 2970,E2 2970} C_VEL
LIN {X 0,Y 562.762,Z 970.096,A -85,B 0,C 180,E1 2973.857,E2 2973.857} C_VEL
LIN {X 0,Y 562.792,Z 961.475,A -85,B 0,C 180,E1 2977.731,E2 2977.731} C_VEL
LIN {X 0,Y 562.938,Z 948.442,A -85,B 0,C 180,E1 2981.209,E2 2981.209} C_VEL
LIN {X 0,Y 563.392,Z 929.156,A -85,B 0,C 180,E1 2984.766,E2 2984.766} C_VEL
LIN {X 0,Y 564.017,Z 904.73,A -85,B 0,C 180,E1 2988.027,E2 2988.027} C_VEL
LIN {X 0,Y 564.895,Z 875.813,A -85,B 0,C 180,E1 2990.905,E2 2990.905} C_VEL
LIN {X 0,Y 565.911,Z 843.22,A -85,B 0,C 180,E1 2993.285,E2 2993.285} C_VEL
LIN {X 0,Y 566.923,Z 809.529,A -85,B 0,C 180,E1 2995.04,E2 2995.04} C_VEL
LIN {X 0,Y 567.703,Z 773.43,A -85,B 0,C 180,E1 2996.27,E2 2996.27} C_VEL
LIN {X 0,Y 567.237,Z 746.845,A -85,B 0,C 180,E1 2996.835,E2 2996.835} C_VEL
LIN {X 0,Y 562.409,Z 733.66,A -85,B 0,C 180,E1 2997.324,E2 2997.324} C_VEL
LIN {X 0,Y 562.094,Z 733.66,A -85,B 0,C 180,E1 3003.379,E2 3003.379} C_VEL
LIN {X 0,Y 561.939,Z 733.66,A -85,B 0,C 180,E1 3008.612,E2 3008.612} C_VEL
LIN {X 0,Y 561.982,Z 733.66,A -85,B 0,C 180,E1 3014.467,E2 3014.467} C_VEL
LIN {X 0,Y 561.988,Z 733.66,A -85,B 0,C 180,E1 3019.712,E2 3019.712} C_VEL
LIN {X 0,Y 561.987,Z 733.66,A -85,B 0,C 180,E1 3025.542,E2 3025.542} C_VEL
LIN {X 0,Y 562.04,Z 733.66,A -85,B 0,C 180,E1 3030.992,E2 3030.992} C_VEL
LIN {X 0,Y 562.209,Z 733.66,A -85,B 0,C 180,E1 3036.3,E2 3036.3} C_VEL
LIN {X 0,Y 562.342,Z 733.66,A -85,B 0,C 180,E1 3041.147,E2 3041.147} C_VEL
LIN {X 0,Y 561.958,Z 733.66,A -85,B 0,C 180,E1 3045.964,E2 3045.964} C_VEL
LIN {X 0,Y 562.284,Z 733.66,A -85,B 0,C 180,E1 3050.699,E2 3050.699} C_VEL
LIN {X 0,Y 562.348,Z 733.66,A -85,B 0,C 180,E1 3055.364,E2 3055.364} C_VEL
LIN {X 0,Y 562.415,Z 733.66,A -85,B 0,C 180,E1 3059.997,E2 3059.997} C_VEL
LIN {X 0,Y 562.346,Z 733.66,A -85,B 0,C 180,E1 3064.988,E2 3064.988} C_VEL
LIN {X 0,Y 562.299,Z 733.66,A -85,B 0,C 180,E1 3070.86,E2 3070.86} C_VEL
LIN {X 0,Y 562.241,Z 733.66,A -85,B 0,C 180,E1 3074.637,E2 3074.637} C_VEL
LIN {X 0,Y 558.251,Z 733.66,A -85,B 0,C 180,E1 3076.381,E2 3076.381} C_VEL
LIN {X 0,Y 554.329,Z 733.66,A -85,B 0,C 180,E1 3078.15,E2 3078.15} C_VEL
LIN {X 0,Y 554.239,Z 733.66,A -85,B 0,C 180,E1 3084.185,E2 3084.185} C_VEL
LIN {X 0,Y 554.162,Z 733.66,A -85,B 0,C 180,E1 3089.453,E2 3089.453} C_VEL
LIN {X 0,Y 554.091,Z 733.66,A -85,B 0,C 180,E1 3095.012,E2 3095.012} C_VEL
LIN {X 0,Y 554.033,Z 733.66,A -85,B 0,C 180,E1 3100.979,E2 3100.979} C_VEL
LIN {X 0,Y 554.166,Z 733.66,A -85,B 0,C 180,E1 3106.917,E2 3106.917} C_VEL
LIN {X 0,Y 554.122,Z 733.66,A -85,B 0,C 180,E1 3113.049,E2 3113.049} C_VEL
LIN {X 0,Y 554.116,Z 733.66,A -85,B 0,C 180,E1 3118.723,E2 3118.723} C_VEL
LIN {X 0,Y 554.261,Z 734.446,A -85,B 0,C 180,E1 3120.006,E2 3120.006} C_VEL
LIN {X 0,Y 556.276,Z 738.929,A -85,B 0,C 180,E1 3121.115,E2 3121.115} C_VEL
LIN {X 0,Y 556.64,Z 740.48,A -85,B 0,C 180,E1 3121.729,E2 3121.729} C_VEL
LIN {X 0,Y 561.064,Z 752.891,A -85,B 0,C 180,E1 3122.178,E2 3122.178} C_VEL
LIN {X 0,Y 560.67,Z 819.649,A -85,B 0,C 180,E1 3123.231,E2 3123.231} C_VEL
LIN {X 0,Y 559.754,Z 856.35,A -85,B 0,C 180,E1 3124.427,E2 3124.427} C_VEL
LIN {X 0,Y 558.599,Z 892.321,A -85,B 0,C 180,E1 3126.285,E2 3126.285} C_VEL
LIN {X 0,Y 557.425,Z 925.124,A -85,B 0,C 180,E1 3128.697,E2 3128.697} C_VEL
LIN {X 0,Y 556.387,Z 953.467,A -85,B 0,C 180,E1 3131.526,E2 3131.526} C_VEL
LIN {X 0,Y 555.622,Z 977.196,A -85,B 0,C 180,E1 3134.672,E2 3134.672} C_VEL
LIN {X 0,Y 555.097,Z 996.69,A -85,B 0,C 180,E1 3138.195,E2 3138.195} C_VEL
LIN {X 0,Y 554.899,Z 1010.436,A -85,B 0,C 180,E1 3141.764,E2 3141.764} C_VEL
LIN {X 0,Y 554.759,Z 1018.964,A -85,B 0,C 180,E1 3145.303,E2 3145.303} C_VEL
LIN {X 0,Y 554.72,Z 1022.523,A -85,B 0,C 180,E1 3148.436,E2 3148.436} C_VEL
LIN {X 0,Y 554.791,Z 1022.522,A -85,B 0,C 180,E1 3151.564,E2 3151.564} C_VEL
LIN {X 0,Y 554.852,Z 1018.962,A -85,B 0,C 180,E1 3154.696,E2 3154.696} C_VEL
LIN {X 0,Y 554.938,Z 1009.194,A -85,B 0,C 180,E1 3158.63,E2 3158.63} C_VEL
LIN {X 0,Y 555.151,Z 994.785,A -85,B 0,C 180,E1 3162.202,E2 3162.202} C_VEL
LIN {X 0,Y 555.668,Z 975.552,A -85,B 0,C 180,E1 3165.575,E2 3165.575} C_VEL
LIN {X 0,Y 556.475,Z 950.122,A -85,B 0,C 180,E1 3168.862,E2 3168.862} C_VEL
LIN {X 0,Y 557.584,Z 920.224,A -85,B 0,C 180,E1 3171.714,E2 3171.714} C_VEL
LIN {X 0,Y 558.817,Z 887.908,A -85,B 0,C 180,E1 3173.98,E2 3173.98} C_VEL
LIN {X 0,Y 559.914,Z 852.458,A -85,B 0,C 180,E1 3175.727,E2 3175.727} C_VEL
LIN {X 0,Y 560.708,Z 815.46,A -85,B 0,C 180,E1 3176.869,E2 3176.869} C_VEL
LIN {X 0,Y 560.568,Z 750.156,A -85,B 0,C 180,E1 3177.888,E2 3177.888} C_VEL
LIN {X 0,Y 556.745,Z 739.944,A -85,B 0,C 180,E1 3178.344,E2 3178.344} C_VEL
LIN {X 0,Y 554.524,Z 735.837,A -85,B 0,C 180,E1 3179.797,E2 3179.797} C_VEL
LIN {X 0,Y 554.217,Z 733.66,A -85,B 0,C 180,E1 3180.176,E2 3180.176} C_VEL
LIN {X 0,Y 554.081,Z 733.66,A -85,B 0,C 180,E1 3185.019,E2 3185.019} C_VEL
LIN {X 0,Y 554.127,Z 733.66,A -85,B 0,C 180,E1 3190.978,E2 3190.978} C_VEL
LIN {X 0,Y 554.069,Z 733.66,A -85,B 0,C 180,E1 3196.916,E2 3196.916} C_VEL
LIN {X 0,Y 554.017,Z 733.66,A -85,B 0,C 180,E1 3203.048,E2 3203.048} C_VEL
LIN {X 0,Y 554.212,Z 733.66,A -85,B 0,C 180,E1 3208.736,E2 3208.736} C_VEL
LIN {X 0,Y 554.13,Z 733.66,A -85,B 0,C 180,E1 3214.38,E2 3214.38} C_VEL
LIN {X 0,Y 554.424,Z 733.66,A -85,B 0,C 180,E1 3220.724,E2 3220.724} C_VEL
LIN {X 0,Y 556.898,Z 751.716,A -85,B 0,C 180,E1 3221.146,E2 3221.146} C_VEL
LIN {X 0,Y 556.518,Z 780.019,A -85,B 0,C 180,E1 3222.132,E2 3222.132} C_VEL
LIN {X 0,Y 556.038,Z 806.385,A -85,B 0,C 180,E1 3223.696,E2 3223.696} C_VEL
LIN {X 0,Y 555.528,Z 829.85,A -85,B 0,C 180,E1 3225.805,E2 3225.805} C_VEL
LIN {X 0,Y 555.161,Z 848.012,A -85,B 0,C 180,E1 3228.201,E2 3228.201} C_VEL
LIN {X 0,Y 554.956,Z 861.788,A -85,B 0,C 180,E1 3230.978,E2 3230.978} C_VEL
LIN {X 0,Y 554.894,Z 869.841,A -85,B 0,C 180,E1 3233.738,E2 3233.738} C_VEL
LIN {X 0,Y 554.791,Z 872.926,A -85,B 0,C 180,E1 3236.875,E2 3236.875} C_VEL
LIN {X 0,Y 554.864,Z 870.171,A -85,B 0,C 180,E1 3240.004,E2 3240.004} C_VEL
LIN {X 0,Y 554.923,Z 862.551,A -85,B 0,C 180,E1 3242.74,E2 3242.74} C_VEL
LIN {X 0,Y 555.18,Z 848.125,A -85,B 0,C 180,E1 3245.689,E2 3245.689} C_VEL
LIN {X 0,Y 555.484,Z 830.538,A -85,B 0,C 180,E1 3248.033,E2 3248.033} C_VEL
LIN {X 0,Y 555.991,Z 806.597,A -85,B 0,C 180,E1 3250.199,E2 3250.199} C_VEL
LIN {X 0,Y 556.604,Z 780.221,A -85,B 0,C 180,E1 3251.761,E2 3251.761} C_VEL
LIN {X 0,Y 557.058,Z 750.654,A -85,B 0,C 180,E1 3252.783,E2 3252.783} C_VEL
LIN {X 0,Y 554.495,Z 733.66,A -85,B 0,C 180,E1 3253.193,E2 3253.193} C_VEL
LIN {X 0,Y 554.336,Z 733.66,A -85,B 0,C 180,E1 3259.136,E2 3259.136} C_VEL
LIN {X 0,Y 554.215,Z 733.66,A -85,B 0,C 180,E1 3264.194,E2 3264.194} C_VEL
LIN {X 0,Y 554.125,Z 733.66,A -85,B 0,C 180,E1 3269.463,E2 3269.463} C_VEL
LIN {X 0,Y 554.106,Z 733.66,A -85,B 0,C 180,E1 3275.019,E2 3275.019} C_VEL
LIN {X 0,Y 554.033,Z 733.66,A -85,B 0,C 180,E1 3280.989,E2 3280.989} C_VEL
LIN {X 0,Y 554.177,Z 733.66,A -85,B 0,C 180,E1 3286.919,E2 3286.919} C_VEL
LIN {X 0,Y 554.095,Z 733.66,A -85,B 0,C 180,E1 3293.047,E2 3293.047} C_VEL
LIN {X 0,Y 554.079,Z 733.66,A -85,B 0,C 180,E1 3298.722,E2 3298.722} C_VEL
LIN {X 0,Y 554.188,Z 733.66,A -85,B 0,C 180,E1 3302.199,E2 3302.199} C_VEL
LIN {X 0,Y 560.789,Z 752.405,A -85,B 0,C 180,E1 3302.831,E2 3302.831} C_VEL
LIN {X 0,Y 560.186,Z 790.318,A -85,B 0,C 180,E1 3303.782,E2 3303.782} C_VEL
LIN {X 0,Y 559.157,Z 827.407,A -85,B 0,C 180,E1 3305.383,E2 3305.383} C_VEL
LIN {X 0,Y 557.863,Z 861.739,A -85,B 0,C 180,E1 3307.575,E2 3307.575} C_VEL
LIN {X 0,Y 556.779,Z 892.842,A -85,B 0,C 180,E1 3310.317,E2 3310.317} C_VEL
LIN {X 0,Y 555.863,Z 918.607,A -85,B 0,C 180,E1 3313.381,E2 3313.381} C_VEL
LIN {X 0,Y 555.333,Z 939.957,A -85,B 0,C 180,E1 3316.801,E2 3316.801} C_VEL
LIN {X 0,Y 554.965,Z 956.655,A -85,B 0,C 180,E1 3320.579,E2 3320.579} C_VEL
LIN {X 0,Y 554.86,Z 965.871,A -85,B 0,C 180,E1 3323.734,E2 3323.734} C_VEL
LIN {X 0,Y 554.806,Z 971.217,A -85,B 0,C 180,E1 3326.871,E2 3326.871} C_VEL
LIN {X 0,Y 554.767,Z 972.997,A -85,B 0,C 180,E1 3330,E2 3330} C_VEL
LIN {X 0,Y 554.881,Z 970.098,A -85,B 0,C 180,E1 3333.912,E2 3333.912} C_VEL
LIN {X 0,Y 554.897,Z 961.478,A -85,B 0,C 180,E1 3337.842,E2 3337.842} C_VEL
LIN {X 0,Y 555.085,Z 948.288,A -85,B 0,C 180,E1 3341.406,E2 3341.406} C_VEL
LIN {X 0,Y 555.605,Z 928.426,A -85,B 0,C 180,E1 3345.09,E2 3345.09} C_VEL
LIN {X 0,Y 556.339,Z 904.784,A -85,B 0,C 180,E1 3348.279,E2 3348.279} C_VEL
LIN {X 0,Y 557.388,Z 875.822,A -85,B 0,C 180,E1 3351.2,E2 3351.2} C_VEL
LIN {X 0,Y 558.571,Z 843.135,A -85,B 0,C 180,E1 3353.615,E2 3353.615} C_VEL
LIN {X 0,Y 559.782,Z 808.874,A -85,B 0,C 180,E1 3355.412,E2 3355.412} C_VEL
LIN {X 0,Y 560.663,Z 772.331,A -85,B 0,C 180,E1 3356.657,E2 3356.657} C_VEL
LIN {X 0,Y 560.11,Z 748.586,A -85,B 0,C 180,E1 3357.179,E2 3357.179} C_VEL
LIN {X 0,Y 554.391,Z 733.66,A -85,B 0,C 180,E1 3357.753,E2 3357.753} C_VEL
LIN {X 0,Y 554.184,Z 733.66,A -85,B 0,C 180,E1 3363.122,E2 3363.122} C_VEL
LIN {X 0,Y 554.015,Z 733.66,A -85,B 0,C 180,E1 3368.946,E2 3368.946} C_VEL
LIN {X 0,Y 554.105,Z 733.66,A -85,B 0,C 180,E1 3374.727,E2 3374.727} C_VEL
LIN {X 0,Y 554.065,Z 733.66,A -85,B 0,C 180,E1 3379.921,E2 3379.921} C_VEL
LIN {X 0,Y 554.066,Z 733.66,A -85,B 0,C 180,E1 3385.066,E2 3385.066} C_VEL
LIN {X 0,Y 554.165,Z 733.66,A -85,B 0,C 180,E1 3390.964,E2 3390.964} C_VEL
LIN {X 0,Y 554.276,Z 733.66,A -85,B 0,C 180,E1 3395.809,E2 3395.809} C_VEL
LIN {X 0,Y 554.429,Z 733.66,A -85,B 0,C 180,E1 3400.868,E2 3400.868} C_VEL
LIN {X 0,Y 554.084,Z 733.66,A -85,B 0,C 180,E1 3405.76,E2 3405.76} C_VEL
LIN {X 0,Y 554.371,Z 733.66,A -85,B 0,C 180,E1 3410.565,E2 3410.565} C_VEL
LIN {X 0,Y 554.471,Z 733.66,A -85,B 0,C 180,E1 3415.298,E2 3415.298} C_VEL
LIN {X 0,Y 554.514,Z 733.66,A -85,B 0,C 180,E1 3419.996,E2 3419.996} C_VEL
LIN {X 0,Y 554.514,Z 733.66,A -85,B 0,C 180,E1 3424.695,E2 3424.695} C_VEL
LIN {X 0,Y 554.383,Z 733.66,A -85,B 0,C 180,E1 3430.513,E2 3430.513} C_VEL
LIN {X 0,Y 554.292,Z 733.66,A -85,B 0,C 180,E1 3435.848,E2 3435.848} C_VEL
LIN {X 0,Y 554.329,Z 733.66,A -85,B 0,C 180,E1 3438.15,E2 3438.15} C_VEL
LIN {X 0,Y 553.06,Z 733.66,A -85,B 0,C 180,E1 3439.042,E2 3439.042} C_VEL
LIN {X 0,Y 546.425,Z 733.66,A -85,B 0,C 180,E1 3441.472,E2 3441.472} C_VEL
LIN {X 0,Y 546.317,Z 733.66,A -85,B 0,C 180,E1 3441.702,E2 3441.702} C_VEL
LIN {X 0,Y 546.297,Z 733.66,A -85,B 0,C 180,E1 3447.513,E2 3447.513} C_VEL
LIN {X 0,Y 546.191,Z 733.66,A -85,B 0,C 180,E1 3453.733,E2 3453.733} C_VEL
LIN {X 0,Y 546.096,Z 733.66,A -85,B 0,C 180,E1 3459.613,E2 3459.613} C_VEL
LIN {X 0,Y 546.203,Z 733.66,A -85,B 0,C 180,E1 3466.131,E2 3466.131} C_VEL
LIN {X 0,Y 546.22,Z 733.66,A -85,B 0,C 180,E1 3472.423,E2 3472.423} C_VEL
LIN {X 0,Y 546.254,Z 734.022,A -85,B 0,C 180,E1 3479.019,E2 3479.019} C_VEL
LIN {X 0,Y 550.38,Z 742.798,A -85,B 0,C 180,E1 3480.157,E2 3480.157} C_VEL
LIN {X 0,Y 553.587,Z 746.767,A -85,B 0,C 180,E1 3481.271,E2 3481.271} C_VEL
LIN {X 0,Y 553.633,Z 752.405,A -85,B 0,C 180,E1 3481.764,E2 3481.764} C_VEL
LIN {X 0,Y 553.62,Z 819.972,A -85,B 0,C 180,E1 3482.871,E2 3482.871} C_VEL
LIN {X 0,Y 552.576,Z 856.184,A -85,B 0,C 180,E1 3484.064,E2 3484.064} C_VEL
LIN {X 0,Y 551.285,Z 891.325,A -85,B 0,C 180,E1 3485.887,E2 3485.887} C_VEL
LIN {X 0,Y 549.948,Z 923.932,A -85,B 0,C 180,E1 3488.287,E2 3488.287} C_VEL
LIN {X 0,Y 548.8,Z 951.983,A -85,B 0,C 180,E1 3491.084,E2 3491.084} C_VEL
LIN {X 0,Y 547.885,Z 976.561,A -85,B 0,C 180,E1 3494.352,E2 3494.352} C_VEL
LIN {X 0,Y 547.248,Z 996.686,A -85,B 0,C 180,E1 3498.024,E2 3498.024} C_VEL
LIN {X 0,Y 547.036,Z 1010.432,A -85,B 0,C 180,E1 3501.645,E2 3501.645} C_VEL
LIN {X 0,Y 546.862,Z 1019.047,A -85,B 0,C 180,E1 3505.282,E2 3505.282} C_VEL
LIN {X 0,Y 546.818,Z 1022.525,A -85,B 0,C 180,E1 3508.413,E2 3508.413} C_VEL
LIN {X 0,Y 546.887,Z 1022.525,A -85,B 0,C 180,E1 3511.586,E2 3511.586} C_VEL
LIN {X 0,Y 546.909,Z 1017.621,A -85,B 0,C 180,E1 3515.481,E2 3515.481} C_VEL
LIN {X 0,Y 547.022,Z 1007.858,A -85,B 0,C 180,E1 3519.158,E2 3519.158} C_VEL
LIN {X 0,Y 547.377,Z 991.846,A -85,B 0,C 180,E1 3522.988,E2 3522.988} C_VEL
LIN {X 0,Y 548.019,Z 969.768,A -85,B 0,C 180,E1 3526.657,E2 3526.657} C_VEL
LIN {X 0,Y 549.106,Z 943.076,A -85,B 0,C 180,E1 3529.892,E2 3529.892} C_VEL
LIN {X 0,Y 550.457,Z 912.39,A -85,B 0,C 180,E1 3532.649,E2 3532.649} C_VEL
LIN {X 0,Y 551.841,Z 879.474,A -85,B 0,C 180,E1 3534.802,E2 3534.802} C_VEL
LIN {X 0,Y 552.987,Z 845.149,A -85,B 0,C 180,E1 3536.364,E2 3536.364} C_VEL
LIN {X 0,Y 553.86,Z 808.633,A -85,B 0,C 180,E1 3537.376,E2 3537.376} C_VEL
LIN {X 0,Y 553.511,Z 752.119,A -85,B 0,C 180,E1 3538.247,E2 3538.247} C_VEL
LIN {X 0,Y 553.298,Z 746.255,A -85,B 0,C 180,E1 3538.888,E2 3538.888} C_VEL
LIN {X 0,Y 549.725,Z 741.658,A -85,B 0,C 180,E1 3540.036,E2 3540.036} C_VEL
LIN {X 0,Y 546.231,Z 733.66,A -85,B 0,C 180,E1 3541.048,E2 3541.048} C_VEL
LIN {X 0,Y 546.195,Z 733.66,A -85,B 0,C 180,E1 3547.579,E2 3547.579} C_VEL
LIN {X 0,Y 546.199,Z 733.66,A -85,B 0,C 180,E1 3553.893,E2 3553.893} C_VEL
LIN {X 0,Y 546.132,Z 733.66,A -85,B 0,C 180,E1 3560.39,E2 3560.39} C_VEL
LIN {X 0,Y 546.234,Z 733.66,A -85,B 0,C 180,E1 3566.339,E2 3566.339} C_VEL
LIN {X 0,Y 546.214,Z 733.66,A -85,B 0,C 180,E1 3571.891,E2 3571.891} C_VEL
LIN {X 0,Y 546.214,Z 733.66,A -85,B 0,C 180,E1 3577.17,E2 3577.17} C_VEL
LIN {X 0,Y 546.5,Z 733.66,A -85,B 0,C 180,E1 3580.461,E2 3580.461} C_VEL
LIN {X 0,Y 549.383,Z 752.16,A -85,B 0,C 180,E1 3580.901,E2 3580.901} C_VEL
LIN {X 0,Y 549.007,Z 781.171,A -85,B 0,C 180,E1 3581.914,E2 3581.914} C_VEL
LIN {X 0,Y 548.428,Z 806.903,A -85,B 0,C 180,E1 3583.463,E2 3583.463} C_VEL
LIN {X 0,Y 547.791,Z 829.904,A -85,B 0,C 180,E1 3585.6,E2 3585.6} C_VEL
LIN {X 0,Y 547.3,Z 847.739,A -85,B 0,C 180,E1 3588.029,E2 3588.029} C_VEL
LIN {X 0,Y 547.091,Z 861.604,A -85,B 0,C 180,E1 3590.848,E2 3590.848} C_VEL
LIN {X 0,Y 546.999,Z 869.748,A -85,B 0,C 180,E1 3593.647,E2 3593.647} C_VEL
LIN {X 0,Y 546.98,Z 872.108,A -85,B 0,C 180,E1 3595.24,E2 3595.24} C_VEL
LIN {X 0,Y 546.921,Z 872.297,A -85,B 0,C 180,E1 3598.417,E2 3598.417} C_VEL
LIN {X 0,Y 547.069,Z 868.531,A -85,B 0,C 180,E1 3600.796,E2 3600.796} C_VEL
LIN {X 0,Y 547.143,Z 859.6,A -85,B 0,C 180,E1 3603.573,E2 3603.573} C_VEL
LIN {X 0,Y 547.394,Z 844.629,A -85,B 0,C 180,E1 3606.355,E2 3606.355} C_VEL
LIN {X 0,Y 547.859,Z 825.724,A -85,B 0,C 180,E1 3608.746,E2 3608.746} C_VEL
LIN {X 0,Y 548.468,Z 802.348,A -85,B 0,C 180,E1 3610.742,E2 3610.742} C_VEL
LIN {X 0,Y 549.129,Z 775.66,A -85,B 0,C 180,E1 3612.217,E2 3612.217} C_VEL
LIN {X 0,Y 549.424,Z 746.824,A -85,B 0,C 180,E1 3613.109,E2 3613.109} C_VEL
LIN {X 0,Y 546.561,Z 733.66,A -85,B 0,C 180,E1 3613.456,E2 3613.456} C_VEL
LIN {X 0,Y 546.404,Z 733.66,A -85,B 0,C 180,E1 3619.586,E2 3619.586} C_VEL
LIN {X 0,Y 546.299,Z 733.66,A -85,B 0,C 180,E1 3624.568,E2 3624.568} C_VEL
LIN {X 0,Y 546.163,Z 733.66,A -85,B 0,C 180,E1 3629.936,E2 3629.936} C_VEL
LIN {X 0,Y 546.114,Z 733.66,A -85,B 0,C 180,E1 3635.609,E2 3635.609} C_VEL
LIN {X 0,Y 546.132,Z 733.66,A -85,B 0,C 180,E1 3641.713,E2 3641.713} C_VEL
LIN {X 0,Y 546.232,Z 733.66,A -85,B 0,C 180,E1 3646.134,E2 3646.134} C_VEL
LIN {X 0,Y 546.197,Z 733.66,A -85,B 0,C 180,E1 3652.421,E2 3652.421} C_VEL
LIN {X 0,Y 546.157,Z 733.66,A -85,B 0,C 180,E1 3658.215,E2 3658.215} C_VEL
LIN {X 0,Y 546.256,Z 733.66,A -85,B 0,C 180,E1 3661.759,E2 3661.759} C_VEL
LIN {X 0,Y 553.724,Z 754.766,A -85,B 0,C 180,E1 3662.5,E2 3662.5} C_VEL
LIN {X 0,Y 552.985,Z 793.451,A -85,B 0,C 180,E1 3663.524,E2 3663.524} C_VEL
LIN {X 0,Y 551.83,Z 829.16,A -85,B 0,C 180,E1 3665.136,E2 3665.136} C_VEL
LIN {X 0,Y 550.382,Z 862.941,A -85,B 0,C 180,E1 3667.348,E2 3667.348} C_VEL
LIN {X 0,Y 549.136,Z 893.615,A -85,B 0,C 180,E1 3670.116,E2 3670.116} C_VEL
LIN {X 0,Y 548.069,Z 920.058,A -85,B 0,C 180,E1 3673.345,E2 3673.345} C_VEL
LIN {X 0,Y 547.406,Z 942.064,A -85,B 0,C 180,E1 3677.013,E2 3677.013} C_VEL
LIN {X 0,Y 547.064,Z 957.993,A -85,B 0,C 180,E1 3680.843,E2 3680.843} C_VEL
LIN {X 0,Y 546.867,Z 967.54,A -85,B 0,C 180,E1 3684.439,E2 3684.439} C_VEL
LIN {X 0,Y 546.809,Z 972.537,A -85,B 0,C 180,E1 3688.414,E2 3688.414} C_VEL
LIN {X 0,Y 546.858,Z 972.48,A -85,B 0,C 180,E1 3691.587,E2 3691.587} C_VEL
LIN {X 0,Y 546.88,Z 968.899,A -85,B 0,C 180,E1 3694.765,E2 3694.765} C_VEL
LIN {X 0,Y 547.035,Z 960.333,A -85,B 0,C 180,E1 3698.355,E2 3698.355} C_VEL
LIN {X 0,Y 547.214,Z 946.495,A -85,B 0,C 180,E1 3701.977,E2 3701.977} C_VEL
LIN {X 0,Y 547.817,Z 927.467,A -85,B 0,C 180,E1 3705.461,E2 3705.461} C_VEL
LIN {X 0,Y 548.735,Z 903.384,A -85,B 0,C 180,E1 3708.709,E2 3708.709} C_VEL
LIN {X 0,Y 549.999,Z 873.385,A -85,B 0,C 180,E1 3711.711,E2 3711.711} C_VEL
LIN {X 0,Y 551.276,Z 842.232,A -85,B 0,C 180,E1 3714.006,E2 3714.006} C_VEL
LIN {X 0,Y 552.611,Z 808.332,A -85,B 0,C 180,E1 3715.791,E2 3715.791} C_VEL
LIN {X 0,Y 553.613,Z 771.3,A -85,B 0,C 180,E1 3717.053,E2 3717.053} C_VEL
LIN {X 0,Y 553.201,Z 751.044,A -85,B 0,C 180,E1 3717.507,E2 3717.507} C_VEL
LIN {X 0,Y 546.418,Z 733.66,A -85,B 0,C 180,E1 3718.187,E2 3718.187} C_VEL
LIN {X 0,Y 546.2,Z 733.66,A -85,B 0,C 180,E1 3723.733,E2 3723.733} C_VEL
LIN {X 0,Y 546.103,Z 733.66,A -85,B 0,C 180,E1 3729.62,E2 3729.62} C_VEL
LIN {X 0,Y 546.184,Z 733.66,A -85,B 0,C 180,E1 3736.128,E2 3736.128} C_VEL
LIN {X 0,Y 546.182,Z 733.66,A -85,B 0,C 180,E1 3742.418,E2 3742.418} C_VEL
LIN {X 0,Y 546.151,Z 733.66,A -85,B 0,C 180,E1 3748.213,E2 3748.213} C_VEL
LIN {X 0,Y 546.323,Z 733.66,A -85,B 0,C 180,E1 3753.675,E2 3753.675} C_VEL
LIN {X 0,Y 546.447,Z 733.66,A -85,B 0,C 180,E1 3758.885,E2 3758.885} C_VEL
LIN {X 0,Y 546.418,Z 733.66,A -85,B 0,C 180,E1 3763.91,E2 3763.91} C_VEL
LIN {X 0,Y 546.472,Z 733.66,A -85,B 0,C 180,E1 3770.428,E2 3770.428} C_VEL
LIN {X 0,Y 546.598,Z 733.66,A -85,B 0,C 180,E1 3775.23,E2 3775.23} C_VEL
LIN {X 0,Y 546.613,Z 733.66,A -85,B 0,C 180,E1 3779.996,E2 3779.996} C_VEL
LIN {X 0,Y 546.612,Z 733.66,A -85,B 0,C 180,E1 3784.763,E2 3784.763} C_VEL
LIN {X 0,Y 546.545,Z 733.66,A -85,B 0,C 180,E1 3789.564,E2 3789.564} C_VEL
LIN {X 0,Y 546.486,Z 733.66,A -85,B 0,C 180,E1 3794.435,E2 3794.435} C_VEL
LIN {X 0,Y 546.432,Z 733.66,A -85,B 0,C 180,E1 3799.593,E2 3799.593} C_VEL
LIN {X 0,Y 546.317,Z 733.66,A -85,B 0,C 180,E1 3801.702,E2 3801.702} C_VEL
LIN {X 0,Y 542.314,Z 733.66,A -85,B 0,C 180,E1 3803.489,E2 3803.489} C_VEL
LIN {X 0,Y 538.328,Z 733.66,A -85,B 0,C 180,E1 3805.302,E2 3805.302} C_VEL
LIN {X 0,Y 538.271,Z 733.66,A -85,B 0,C 180,E1 3810.413,E2 3810.413} C_VEL
LIN {X 0,Y 538.172,Z 733.66,A -85,B 0,C 180,E1 3816.208,E2 3816.208} C_VEL
LIN {X 0,Y 538.147,Z 733.66,A -85,B 0,C 180,E1 3822.465,E2 3822.465} C_VEL
LIN {X 0,Y 538.228,Z 733.66,A -85,B 0,C 180,E1 3827.534,E2 3827.534} C_VEL
LIN {X 0,Y 538.24,Z 733.66,A -85,B 0,C 180,E1 3833.79,E2 3833.79} C_VEL
LIN {X 0,Y 538.343,Z 734.094,A -85,B 0,C 180,E1 3838.575,E2 3838.575} C_VEL
LIN {X 0,Y 541.568,Z 742.985,A -85,B 0,C 180,E1 3839.318,E2 3839.318} C_VEL
LIN {X 0,Y 547.946,Z 751.725,A -85,B 0,C 180,E1 3840.604,E2 3840.604} C_VEL
LIN {X 0,Y 549.079,Z 754.357,A -85,B 0,C 180,E1 3841.041,E2 3841.041} C_VEL
LIN {X 0,Y 547.161,Z 763.301,A -85,B 0,C 180,E1 3841.559,E2 3841.559} C_VEL
LIN {X 0,Y 546.588,Z 820.591,A -85,B 0,C 180,E1 3842.508,E2 3842.508} C_VEL
LIN {X 0,Y 545.388,Z 857.08,A -85,B 0,C 180,E1 3843.735,E2 3843.735} C_VEL
LIN {X 0,Y 543.91,Z 893.008,A -85,B 0,C 180,E1 3845.648,E2 3845.648} C_VEL
LIN {X 0,Y 542.362,Z 926.305,A -85,B 0,C 180,E1 3848.183,E2 3848.183} C_VEL
LIN {X 0,Y 541.089,Z 953.73,A -85,B 0,C 180,E1 3851.016,E2 3851.016} C_VEL
LIN {X 0,Y 540.057,Z 977.997,A -85,B 0,C 180,E1 3854.345,E2 3854.345} C_VEL
LIN {X 0,Y 539.436,Z 996.682,A -85,B 0,C 180,E1 3857.847,E2 3857.847} C_VEL
LIN {X 0,Y 539.15,Z 1010.428,A -85,B 0,C 180,E1 3861.521,E2 3861.521} C_VEL
LIN {X 0,Y 538.969,Z 1018.956,A -85,B 0,C 180,E1 3865.165,E2 3865.165} C_VEL
LIN {X 0,Y 538.931,Z 1022.527,A -85,B 0,C 180,E1 3868.39,E2 3868.39} C_VEL
LIN {X 0,Y 538.996,Z 1022.527,A -85,B 0,C 180,E1 3871.609,E2 3871.609} C_VEL
LIN {X 0,Y 538.996,Z 1017.467,A -85,B 0,C 180,E1 3875.642,E2 3875.642} C_VEL
LIN {X 0,Y 539.139,Z 1007.86,A -85,B 0,C 180,E1 3879.293,E2 3879.293} C_VEL
LIN {X 0,Y 539.541,Z 991.847,A -85,B 0,C 180,E1 3883.18,E2 3883.18} C_VEL
LIN {X 0,Y 540.295,Z 970.111,A -85,B 0,C 180,E1 3886.854,E2 3886.854} C_VEL
LIN {X 0,Y 541.476,Z 943.879,A -85,B 0,C 180,E1 3890.096,E2 3890.096} C_VEL
LIN {X 0,Y 542.99,Z 913.35,A -85,B 0,C 180,E1 3892.903,E2 3892.903} C_VEL
LIN {X 0,Y 544.595,Z 879.473,A -85,B 0,C 180,E1 3895.154,E2 3895.154} C_VEL
LIN {X 0,Y 545.902,Z 844.727,A -85,B 0,C 180,E1 3896.749,E2 3896.749} C_VEL
LIN {X 0,Y 546.863,Z 808.679,A -85,B 0,C 180,E1 3897.755,E2 3897.755} C_VEL
LIN {X 0,Y 547.325,Z 762.16,A -85,B 0,C 180,E1 3898.503,E2 3898.503} C_VEL
LIN {X 0,Y 549.113,Z 754.308,A -85,B 0,C 180,E1 3898.957,E2 3898.957} C_VEL
LIN {X 0,Y 542.69,Z 744.35,A -85,B 0,C 180,E1 3900.514,E2 3900.514} C_VEL
LIN {X 0,Y 538.407,Z 734.737,A -85,B 0,C 180,E1 3901.355,E2 3901.355} C_VEL
LIN {X 0,Y 538.341,Z 733.66,A -85,B 0,C 180,E1 3901.424,E2 3901.424} C_VEL
LIN {X 0,Y 538.259,Z 733.66,A -85,B 0,C 180,E1 3908.046,E2 3908.046} C_VEL
LIN {X 0,Y 538.238,Z 733.66,A -85,B 0,C 180,E1 3913.005,E2 3913.005} C_VEL
LIN {X 0,Y 538.15,Z 733.66,A -85,B 0,C 180,E1 3919.433,E2 3919.433} C_VEL
LIN {X 0,Y 538.256,Z 733.66,A -85,B 0,C 180,E1 3925.771,E2 3925.771} C_VEL
LIN {X 0,Y 538.275,Z 733.66,A -85,B 0,C 180,E1 3931.439,E2 3931.439} C_VEL
LIN {X 0,Y 538.309,Z 733.66,A -85,B 0,C 180,E1 3936.816,E2 3936.816} C_VEL
LIN {X 0,Y 538.539,Z 733.7,A -85,B 0,C 180,E1 3940.222,E2 3940.222} C_VEL
LIN {X 0,Y 541.762,Z 751.173,A -85,B 0,C 180,E1 3940.622,E2 3940.622} C_VEL
LIN {X 0,Y 541.576,Z 779.664,A -85,B 0,C 180,E1 3941.568,E2 3941.568} C_VEL
LIN {X 0,Y 540.906,Z 806.301,A -85,B 0,C 180,E1 3943.122,E2 3943.122} C_VEL
LIN {X 0,Y 540.237,Z 829.532,A -85,B 0,C 180,E1 3945.243,E2 3945.243} C_VEL
LIN {X 0,Y 539.676,Z 847.5,A -85,B 0,C 180,E1 3947.652,E2 3947.652} C_VEL
LIN {X 0,Y 539.301,Z 860.658,A -85,B 0,C 180,E1 3950.306,E2 3950.306} C_VEL
LIN {X 0,Y 539.115,Z 870.016,A -85,B 0,C 180,E1 3953.554,E2 3953.554} C_VEL
LIN {X 0,Y 539.002,Z 873.128,A -85,B 0,C 180,E1 3956.783,E2 3956.783} C_VEL
LIN {X 0,Y 539.074,Z 870.602,A -85,B 0,C 180,E1 3960.004,E2 3960.004} C_VEL
LIN {X 0,Y 539.217,Z 863.398,A -85,B 0,C 180,E1 3962.82,E2 3962.82} C_VEL
LIN {X 0,Y 539.575,Z 849.614,A -85,B 0,C 180,E1 3965.842,E2 3965.842} C_VEL
LIN {X 0,Y 540.02,Z 832.596,A -85,B 0,C 180,E1 3968.265,E2 3968.265} C_VEL
LIN {X 0,Y 540.719,Z 809.359,A -85,B 0,C 180,E1 3970.49,E2 3970.49} C_VEL
LIN {X 0,Y 541.364,Z 784.606,A -85,B 0,C 180,E1 3972.063,E2 3972.063} C_VEL
LIN {X 0,Y 541.882,Z 755.829,A -85,B 0,C 180,E1 3973.145,E2 3973.145} C_VEL
LIN {X 0,Y 540.493,Z 741.438,A -85,B 0,C 180,E1 3973.498,E2 3973.498} C_VEL
LIN {X 0,Y 538.61,Z 733.66,A -85,B 0,C 180,E1 3973.756,E2 3973.756} C_VEL
LIN {X 0,Y 538.499,Z 733.66,A -85,B 0,C 180,E1 3979.721,E2 3979.721} C_VEL
LIN {X 0,Y 538.302,Z 733.66,A -85,B 0,C 180,E1 3985.833,E2 3985.833} C_VEL
LIN {X 0,Y 538.258,Z 733.66,A -85,B 0,C 180,E1 3990.422,E2 3990.422} C_VEL
LIN {X 0,Y 538.188,Z 733.66,A -85,B 0,C 180,E1 3996.216,E2 3996.216} C_VEL
LIN {X 0,Y 538.162,Z 733.66,A -85,B 0,C 180,E1 4002.474,E2 4002.474} C_VEL
LIN {X 0,Y 538.231,Z 733.66,A -85,B 0,C 180,E1 4007.535,E2 4007.535} C_VEL
LIN {X 0,Y 538.225,Z 733.66,A -85,B 0,C 180,E1 4013.79,E2 4013.79} C_VEL
LIN {X 0,Y 538.249,Z 733.66,A -85,B 0,C 180,E1 4019.58,E2 4019.58} C_VEL
LIN {X 0,Y 538.361,Z 733.66,A -85,B 0,C 180,E1 4021.295,E2 4021.295} C_VEL
LIN {X 0,Y 546.68,Z 756.76,A -85,B 0,C 180,E1 4022.153,E2 4022.153} C_VEL
LIN {X 0,Y 545.818,Z 795.83,A -85,B 0,C 180,E1 4023.243,E2 4023.243} C_VEL
LIN {X 0,Y 544.509,Z 830.531,A -85,B 0,C 180,E1 4024.86,E2 4024.86} C_VEL
LIN {X 0,Y 542.908,Z 864.386,A -85,B 0,C 180,E1 4027.134,E2 4027.134} C_VEL
LIN {X 0,Y 541.443,Z 895.495,A -85,B 0,C 180,E1 4030.031,E2 4030.031} C_VEL
LIN {X 0,Y 540.263,Z 921.767,A -85,B 0,C 180,E1 4033.346,E2 4033.346} C_VEL
LIN {X 0,Y 539.542,Z 943.044,A -85,B 0,C 180,E1 4037.027,E2 4037.027} C_VEL
LIN {X 0,Y 539.194,Z 957.992,A -85,B 0,C 180,E1 4040.708,E2 4040.708} C_VEL
LIN {X 0,Y 538.975,Z 967.539,A -85,B 0,C 180,E1 4044.358,E2 4044.358} C_VEL
LIN {X 0,Y 539.014,Z 971.215,A -85,B 0,C 180,E1 4046.78,E2 4046.78} C_VEL
LIN {X 0,Y 538.974,Z 972.997,A -85,B 0,C 180,E1 4050,E2 4050} C_VEL
LIN {X 0,Y 539.062,Z 970.404,A -85,B 0,C 180,E1 4053.821,E2 4053.821} C_VEL
LIN {X 0,Y 539.152,Z 962.624,A -85,B 0,C 180,E1 4057.666,E2 4057.666} C_VEL
LIN {X 0,Y 539.352,Z 950.033,A -85,B 0,C 180,E1 4061.333,E2 4061.333} C_VEL
